LIN {X 0,Y 361.862,Z 339.034,A -85,B 0,C 180,E1 -13100.973,E2 -13100.973} C_VEL
LIN {X 0,Y 361.867,Z 339.03,A -85,B 0,C 180,E1 -13104.655,E2 -13104.655} C_VEL
LIN {X 0,Y 361.829,Z 339.027,A -85,B 0,C 180,E1 -13108.37,E2 -13108.37} C_VEL
LIN {X 0,Y 361.857,Z 339.016,A -85,B 0,C 180,E1 -13110.952,E2 -13110.952} C_VEL
LIN {X 0,Y 361.874,Z 339.028,A -85,B 0,C 180,E1 -13114.706,E2 -13114.706} C_VEL
LIN {X 0,Y 361.851,Z 339.032,A -85,B 0,C 180,E1 -13118.345,E2 -13118.345} C_VEL
LIN {X 0,Y 361.911,Z 339.028,A -85,B 0,C 180,E1 -13122.085,E2 -13122.085} C_VEL
LIN {X 0,Y 361.951,Z 339.022,A -85,B 0,C 180,E1 -13125.38,E2 -13125.38} C_VEL
LIN {X 0,Y 361.95,Z 339.014,A -85,B 0,C 180,E1 -13128.804,E2 -13128.804} C_VEL
LIN {X 0,Y 362.066,Z 339.002,A -85,B 0,C 180,E1 -13132.191,E2 -13132.191} C_VEL
LIN {X 0,Y 362.08,Z 339.004,A -85,B 0,C 180,E1 -13134.431,E2 -13134.431} C_VEL
LIN {X 0,Y 362.253,Z 338.978,A -85,B 0,C 180,E1 -13137.777,E2 -13137.777} C_VEL
LIN {X 0,Y 362.26,Z 338.976,A -85,B 0,C 180,E1 -13142.224,E2 -13142.224} C_VEL
LIN {X 0,Y 362.131,Z 338.998,A -85,B 0,C 180,E1 -13146.687,E2 -13146.687} C_VEL
LIN {X 0,Y 361.989,Z 339.017,A -85,B 0,C 180,E1 -13150.064,E2 -13150.064} C_VEL
LIN {X 0,Y 361.989,Z 339.017,A -85,B 0,C 180,E1 -13153.899,E2 -13153.899} C_VEL
LIN {X 0,Y 361.919,Z 339.022,A -85,B 0,C 180,E1 -13156.935,E2 -13156.935} C_VEL
LIN {X 0,Y 361.875,Z 339.028,A -85,B 0,C 180,E1 -13160.462,E2 -13160.462} C_VEL
LIN {X 0,Y 361.886,Z 339.028,A -85,B 0,C 180,E1 -13164.114,E2 -13164.114} C_VEL
LIN {X 0,Y 361.935,Z 339.028,A -85,B 0,C 180,E1 -13166.722,E2 -13166.722} C_VEL
LIN {X 0,Y 361.867,Z 339.035,A -85,B 0,C 180,E1 -13170.329,E2 -13170.329} C_VEL
LIN {X 0,Y 361.849,Z 339.033,A -85,B 0,C 180,E1 -13174.282,E2 -13174.282} C_VEL
LIN {X 0,Y 361.858,Z 339.029,A -85,B 0,C 180,E1 -13177.224,E2 -13177.224} C_VEL
LIN {X 0,Y 361.831,Z 339.038,A -85,B 0,C 180,E1 -13180.756,E2 -13180.756} C_VEL
LIN {X 0,Y 361.814,Z 339.041,A -85,B 0,C 180,E1 -13184.37,E2 -13184.37} C_VEL
LIN {X 0,Y 361.834,Z 339.039,A -85,B 0,C 180,E1 -13187.569,E2 -13187.569} C_VEL
LIN {X 0,Y 361.87,Z 339.036,A -85,B 0,C 180,E1 -13190.974,E2 -13190.974} C_VEL
LIN {X 0,Y 361.896,Z 339.076,A -85,B 0,C 180,E1 -13193.507,E2 -13193.507} C_VEL
LIN {X 0,Y 364.21,Z 348.551,A -85,B 0,C 180,E1 -13196.226,E2 -13196.226} C_VEL
LIN {X 0,Y 374.313,Z 370.595,A -85,B 0,C 180,E1 -13197.6,E2 -13197.6} C_VEL
LIN {X 0,Y 376.246,Z 375.985,A -85,B 0,C 180,E1 -13197.878,E2 -13197.878} C_VEL
LIN {X 0,Y 377.03,Z 379.634,A -85,B 0,C 180,E1 -13198.02,E2 -13198.02} C_VEL
LIN {X 0,Y 374.531,Z 484.966,A -85,B 0,C 180,E1 -13200.078,E2 -13200.078} C_VEL
LIN {X 0,Y 373.805,Z 499.549,A -85,B 0,C 180,E1 -13200.585,E2 -13200.585} C_VEL
LIN {X 0,Y 372.836,Z 513.064,A -85,B 0,C 180,E1 -13201.271,E2 -13201.271} C_VEL
LIN {X 0,Y 371.435,Z 527.178,A -85,B 0,C 180,E1 -13202.23,E2 -13202.23} C_VEL
LIN {X 0,Y 369.952,Z 539.936,A -85,B 0,C 180,E1 -13203.353,E2 -13203.353} C_VEL
LIN {X 0,Y 368.362,Z 551.192,A -85,B 0,C 180,E1 -13204.579,E2 -13204.579} C_VEL
LIN {X 0,Y 366.879,Z 561.686,A -85,B 0,C 180,E1 -13205.98,E2 -13205.98} C_VEL
LIN {X 0,Y 365.475,Z 572.081,A -85,B 0,C 180,E1 -13207.68,E2 -13207.68} C_VEL
LIN {X 0,Y 364.078,Z 580.622,A -85,B 0,C 180,E1 -13209.373,E2 -13209.373} C_VEL
LIN {X 0,Y 362.866,Z 588.744,A -85,B 0,C 180,E1 -13211.364,E2 -13211.364} C_VEL
LIN {X 0,Y 362.032,Z 594.441,A -85,B 0,C 180,E1 -13213.071,E2 -13213.071} C_VEL
LIN {X 0,Y 361.23,Z 600.377,A -85,B 0,C 180,E1 -13215.35,E2 -13215.35} C_VEL
LIN {X 0,Y 360.7,Z 604.706,A -85,B 0,C 180,E1 -13217.624,E2 -13217.624} C_VEL
LIN {X 0,Y 360.32,Z 607.567,A -85,B 0,C 180,E1 -13219.89,E2 -13219.89} C_VEL
LIN {X 0,Y 360.302,Z 609.048,A -85,B 0,C 180,E1 -13222.152,E2 -13222.152} C_VEL
LIN {X 0,Y 360.342,Z 609.198,A -85,B 0,C 180,E1 -13224.404,E2 -13224.404} C_VEL
LIN {X 0,Y 360.318,Z 608.032,A -85,B 0,C 180,E1 -13226.646,E2 -13226.646} C_VEL
LIN {X 0,Y 360.47,Z 605.531,A -85,B 0,C 180,E1 -13228.883,E2 -13228.883} C_VEL
LIN {X 0,Y 360.675,Z 601.614,A -85,B 0,C 180,E1 -13231.116,E2 -13231.116} C_VEL
LIN {X 0,Y 361.122,Z 596.159,A -85,B 0,C 180,E1 -13233.347,E2 -13233.347} C_VEL
LIN {X 0,Y 361.799,Z 589.999,A -85,B 0,C 180,E1 -13235.294,E2 -13235.294} C_VEL
LIN {X 0,Y 362.798,Z 582.325,A -85,B 0,C 180,E1 -13237.233,E2 -13237.233} C_VEL
LIN {X 0,Y 363.83,Z 574.327,A -85,B 0,C 180,E1 -13238.889,E2 -13238.889} C_VEL
LIN {X 0,Y 364.883,Z 564.682,A -85,B 0,C 180,E1 -13240.548,E2 -13240.548} C_VEL
LIN {X 0,Y 366.129,Z 554.042,A -85,B 0,C 180,E1 -13242.049,E2 -13242.049} C_VEL
LIN {X 0,Y 367.506,Z 542.214,A -85,B 0,C 180,E1 -13243.407,E2 -13243.407} C_VEL
LIN {X 0,Y 368.64,Z 530.605,A -85,B 0,C 180,E1 -13244.49,E2 -13244.49} C_VEL
LIN {X 0,Y 369.853,Z 516.946,A -85,B 0,C 180,E1 -13245.498,E2 -13245.498} C_VEL
LIN {X 0,Y 370.304,Z 510.93,A -85,B 0,C 180,E1 -13245.859,E2 -13245.859} C_VEL
LIN {X 0,Y 370.012,Z 505.422,A -85,B 0,C 180,E1 -13246.193,E2 -13246.193} C_VEL
LIN {X 0,Y 367.793,Z 496.434,A -85,B 0,C 180,E1 -13246.755,E2 -13246.755} C_VEL
LIN {X 0,Y 365.53,Z 487.277,A -85,B 0,C 180,E1 -13247.225,E2 -13247.225} C_VEL
LIN {X 0,Y 365.142,Z 481.513,A -85,B 0,C 180,E1 -13247.408,E2 -13247.408} C_VEL
LIN {X 0,Y 367.072,Z 379.114,A -85,B 0,C 180,E1 -13249.428,E2 -13249.428} C_VEL
LIN {X 0,Y 365.066,Z 369.722,A -85,B 0,C 180,E1 -13249.762,E2 -13249.762} C_VEL
LIN {X 0,Y 357.701,Z 350.958,A -85,B 0,C 180,E1 -13250.685,E2 -13250.685} C_VEL
LIN {X 0,Y 356.686,Z 348.279,A -85,B 0,C 180,E1 -13250.833,E2 -13250.833} C_VEL
LIN {X 0,Y 354.849,Z 339.909,A -85,B 0,C 180,E1 -13253.142,E2 -13253.142} C_VEL
LIN {X 0,Y 354.889,Z 339.904,A -85,B 0,C 180,E1 -13256.98,E2 -13256.98} C_VEL
LIN {X 0,Y 354.819,Z 339.911,A -85,B 0,C 180,E1 -13259.681,E2 -13259.681} C_VEL
LIN {X 0,Y 354.806,Z 339.916,A -85,B 0,C 180,E1 -13263.701,E2 -13263.701} C_VEL
LIN {X 0,Y 354.801,Z 339.91,A -85,B 0,C 180,E1 -13266.458,E2 -13266.458} C_VEL
LIN {X 0,Y 354.823,Z 339.901,A -85,B 0,C 180,E1 -13269.422,E2 -13269.422} C_VEL
LIN {X 0,Y 354.786,Z 339.914,A -85,B 0,C 180,E1 -13272.866,E2 -13272.866} C_VEL
LIN {X 0,Y 354.764,Z 339.918,A -85,B 0,C 180,E1 -13276.102,E2 -13276.102} C_VEL
LIN {X 0,Y 354.783,Z 339.913,A -85,B 0,C 180,E1 -13279.178,E2 -13279.178} C_VEL
LIN {X 0,Y 354.802,Z 339.906,A -85,B 0,C 180,E1 -13282.402,E2 -13282.402} C_VEL
LIN {X 0,Y 354.807,Z 339.915,A -85,B 0,C 180,E1 -13284.94,E2 -13284.94} C_VEL
LIN {X 0,Y 354.787,Z 339.913,A -85,B 0,C 180,E1 -13288.404,E2 -13288.404} C_VEL
LIN {X 0,Y 354.831,Z 339.898,A -85,B 0,C 180,E1 -13291.617,E2 -13291.617} C_VEL
LIN {X 0,Y 354.867,Z 339.899,A -85,B 0,C 180,E1 -13294.17,E2 -13294.17} C_VEL
LIN {X 0,Y 354.8,Z 339.907,A -85,B 0,C 180,E1 -13297.891,E2 -13297.891} C_VEL
LIN {X 0,Y 354.881,Z 339.899,A -85,B 0,C 180,E1 -13301.907,E2 -13301.907} C_VEL
LIN {X 0,Y 354.934,Z 339.888,A -85,B 0,C 180,E1 -13305.981,E2 -13305.981} C_VEL
LIN {X 0,Y 354.945,Z 339.89,A -85,B 0,C 180,E1 -13309.734,E2 -13309.734} C_VEL
LIN {X 0,Y 355.095,Z 339.87,A -85,B 0,C 180,E1 -13313.18,E2 -13313.18} C_VEL
LIN {X 0,Y 355.219,Z 339.855,A -85,B 0,C 180,E1 -13317.732,E2 -13317.732} C_VEL
LIN {X 0,Y 355.159,Z 339.864,A -85,B 0,C 180,E1 -13321.133,E2 -13321.133} C_VEL
LIN {X 0,Y 355.206,Z 339.856,A -85,B 0,C 180,E1 -13322.267,E2 -13322.267} C_VEL
LIN {X 0,Y 355.073,Z 339.879,A -85,B 0,C 180,E1 -13326.82,E2 -13326.82} C_VEL
LIN {X 0,Y 354.943,Z 339.887,A -85,B 0,C 180,E1 -13330.265,E2 -13330.265} C_VEL
LIN {X 0,Y 354.933,Z 339.897,A -85,B 0,C 180,E1 -13334.018,E2 -13334.018} C_VEL
LIN {X 0,Y 354.88,Z 339.904,A -85,B 0,C 180,E1 -13338.092,E2 -13338.092} C_VEL
LIN {X 0,Y 354.805,Z 339.906,A -85,B 0,C 180,E1 -13342.108,E2 -13342.108} C_VEL
LIN {X 0,Y 354.812,Z 339.906,A -85,B 0,C 180,E1 -13345.834,E2 -13345.834} C_VEL
LIN {X 0,Y 354.788,Z 339.914,A -85,B 0,C 180,E1 -13349.684,E2 -13349.684} C_VEL
LIN {X 0,Y 354.778,Z 339.917,A -85,B 0,C 180,E1 -13352.334,E2 -13352.334} C_VEL
LIN {X 0,Y 354.814,Z 339.914,A -85,B 0,C 180,E1 -13355.7,E2 -13355.7} C_VEL
LIN {X 0,Y 354.817,Z 339.913,A -85,B 0,C 180,E1 -13359.424,E2 -13359.424} C_VEL
LIN {X 0,Y 354.782,Z 339.912,A -85,B 0,C 180,E1 -13362.868,E2 -13362.868} C_VEL
LIN {X 0,Y 354.761,Z 339.919,A -85,B 0,C 180,E1 -13366.104,E2 -13366.104} C_VEL
LIN {X 0,Y 354.782,Z 339.918,A -85,B 0,C 180,E1 -13369.18,E2 -13369.18} C_VEL
LIN {X 0,Y 354.802,Z 339.918,A -85,B 0,C 180,E1 -13372.403,E2 -13372.403} C_VEL
LIN {X 0,Y 354.808,Z 339.919,A -85,B 0,C 180,E1 -13374.942,E2 -13374.942} C_VEL
LIN {X 0,Y 354.835,Z 340.014,A -85,B 0,C 180,E1 -13377.168,E2 -13377.168} C_VEL
LIN {X 0,Y 358.077,Z 353.914,A -85,B 0,C 180,E1 -13380.616,E2 -13380.616} C_VEL
LIN {X 0,Y 360.084,Z 364.069,A -85,B 0,C 180,E1 -13383.014,E2 -13383.014} C_VEL
LIN {X 0,Y 360.134,Z 366.037,A -85,B 0,C 180,E1 -13383.448,E2 -13383.448} C_VEL
LIN {X 0,Y 365.056,Z 394.772,A -85,B 0,C 180,E1 -13384.402,E2 -13384.402} C_VEL
LIN {X 0,Y 366.748,Z 405.34,A -85,B 0,C 180,E1 -13384.736,E2 -13384.736} C_VEL
LIN {X 0,Y 364.738,Z 503.037,A -85,B 0,C 180,E1 -13386.659,E2 -13386.659} C_VEL
LIN {X 0,Y 364,Z 517.441,A -85,B 0,C 180,E1 -13387.135,E2 -13387.135} C_VEL
LIN {X 0,Y 363.018,Z 531.264,A -85,B 0,C 180,E1 -13387.821,E2 -13387.821} C_VEL
LIN {X 0,Y 361.901,Z 543.849,A -85,B 0,C 180,E1 -13388.655,E2 -13388.655} C_VEL
LIN {X 0,Y 360.585,Z 556.821,A -85,B 0,C 180,E1 -13389.76,E2 -13389.76} C_VEL
LIN {X 0,Y 359.18,Z 568.653,A -85,B 0,C 180,E1 -13391.017,E2 -13391.017} C_VEL
LIN {X 0,Y 357.972,Z 578.49,A -85,B 0,C 180,E1 -13392.284,E2 -13392.284} C_VEL
LIN {X 0,Y 356.588,Z 589.361,A -85,B 0,C 180,E1 -13393.983,E2 -13393.983} C_VEL
LIN {X 0,Y 355.57,Z 598.603,A -85,B 0,C 180,E1 -13395.753,E2 -13395.753} C_VEL
LIN {X 0,Y 354.694,Z 606.928,A -85,B 0,C 180,E1 -13397.702,E2 -13397.702} C_VEL
LIN {X 0,Y 353.92,Z 613.835,A -85,B 0,C 180,E1 -13399.705,E2 -13399.705} C_VEL
LIN {X 0,Y 353.58,Z 618.593,A -85,B 0,C 180,E1 -13401.427,E2 -13401.427} C_VEL
LIN {X 0,Y 353.4,Z 622.44,A -85,B 0,C 180,E1 -13403.147,E2 -13403.147} C_VEL
LIN {X 0,Y 353.269,Z 626.191,A -85,B 0,C 180,E1 -13405.436,E2 -13405.436} C_VEL
LIN {X 0,Y 353.181,Z 628.521,A -85,B 0,C 180,E1 -13407.719,E2 -13407.719} C_VEL
LIN {X 0,Y 353.261,Z 629.496,A -85,B 0,C 180,E1 -13410,E2 -13410} C_VEL
LIN {X 0,Y 353.168,Z 629.129,A -85,B 0,C 180,E1 -13412.281,E2 -13412.281} C_VEL
LIN {X 0,Y 353.246,Z 627.432,A -85,B 0,C 180,E1 -13414.564,E2 -13414.564} C_VEL
LIN {X 0,Y 353.411,Z 624.368,A -85,B 0,C 180,E1 -13416.853,E2 -13416.853} C_VEL
LIN {X 0,Y 353.772,Z 619.856,A -85,B 0,C 180,E1 -13419.144,E2 -13419.144} C_VEL
LIN {X 0,Y 354.219,Z 615.396,A -85,B 0,C 180,E1 -13420.864,E2 -13420.864} C_VEL
LIN {X 0,Y 355.178,Z 608.979,A -85,B 0,C 180,E1 -13422.862,E2 -13422.862} C_VEL
LIN {X 0,Y 356.2,Z 601.025,A -85,B 0,C 180,E1 -13424.862,E2 -13424.862} C_VEL
LIN {X 0,Y 357.49,Z 592.726,A -85,B 0,C 180,E1 -13426.562,E2 -13426.562} C_VEL
LIN {X 0,Y 359.067,Z 582.754,A -85,B 0,C 180,E1 -13428.25,E2 -13428.25} C_VEL
LIN {X 0,Y 360.864,Z 571.675,A -85,B 0,C 180,E1 -13429.778,E2 -13429.778} C_VEL
LIN {X 0,Y 362.613,Z 559.29,A -85,B 0,C 180,E1 -13431.16,E2 -13431.16} C_VEL
LIN {X 0,Y 364.133,Z 547.349,A -85,B 0,C 180,E1 -13432.231,E2 -13432.231} C_VEL
LIN {X 0,Y 365.442,Z 534.552,A -85,B 0,C 180,E1 -13433.143,E2 -13433.143} C_VEL
LIN {X 0,Y 366.783,Z 520.612,A -85,B 0,C 180,E1 -13433.877,E2 -13433.877} C_VEL
LIN {X 0,Y 367.758,Z 505.981,A -85,B 0,C 180,E1 -13434.409,E2 -13434.409} C_VEL
LIN {X 0,Y 368.551,Z 481.48,A -85,B 0,C 180,E1 -13434.928,E2 -13434.928} C_VEL
LIN {X 0,Y 370.194,Z 405.301,A -85,B 0,C 180,E1 -13436.436,E2 -13436.436} C_VEL
LIN {X 0,Y 365.616,Z 381.424,A -85,B 0,C 180,E1 -13437.353,E2 -13437.353} C_VEL
LIN {X 0,Y 362.959,Z 370.452,A -85,B 0,C 180,E1 -13437.836,E2 -13437.836} C_VEL
LIN {X 0,Y 361.045,Z 365.765,A -85,B 0,C 180,E1 -13438.117,E2 -13438.117} C_VEL
LIN {X 0,Y 358.588,Z 354.578,A -85,B 0,C 180,E1 -13440.961,E2 -13440.961} C_VEL
LIN {X 0,Y 355.383,Z 342.059,A -85,B 0,C 180,E1 -13444.354,E2 -13444.354} C_VEL
LIN {X 0,Y 354.869,Z 339.906,A -85,B 0,C 180,E1 -13444.971,E2 -13444.971} C_VEL
LIN {X 0,Y 354.801,Z 339.903,A -85,B 0,C 180,E1 -13447.882,E2 -13447.882} C_VEL
LIN {X 0,Y 354.782,Z 339.904,A -85,B 0,C 180,E1 -13451.171,E2 -13451.171} C_VEL
LIN {X 0,Y 354.758,Z 339.914,A -85,B 0,C 180,E1 -13454.506,E2 -13454.506} C_VEL
LIN {X 0,Y 354.788,Z 339.91,A -85,B 0,C 180,E1 -13457.662,E2 -13457.662} C_VEL
LIN {X 0,Y 354.809,Z 339.914,A -85,B 0,C 180,E1 -13460.665,E2 -13460.665} C_VEL
LIN {X 0,Y 354.814,Z 339.911,A -85,B 0,C 180,E1 -13464.3,E2 -13464.3} C_VEL
LIN {X 0,Y 354.779,Z 339.915,A -85,B 0,C 180,E1 -13467.666,E2 -13467.666} C_VEL
LIN {X 0,Y 354.793,Z 339.9,A -85,B 0,C 180,E1 -13471.614,E2 -13471.614} C_VEL
LIN {X 0,Y 354.825,Z 339.905,A -85,B 0,C 180,E1 -13475.657,E2 -13475.657} C_VEL
LIN {X 0,Y 354.816,Z 339.907,A -85,B 0,C 180,E1 -13479.113,E2 -13479.113} C_VEL
LIN {X 0,Y 354.87,Z 339.902,A -85,B 0,C 180,E1 -13482.719,E2 -13482.719} C_VEL
LIN {X 0,Y 354.941,Z 339.896,A -85,B 0,C 180,E1 -13486.255,E2 -13486.255} C_VEL
LIN {X 0,Y 354.939,Z 339.896,A -85,B 0,C 180,E1 -13489.735,E2 -13489.735} C_VEL
LIN {X 0,Y 355.076,Z 339.871,A -85,B 0,C 180,E1 -13493.18,E2 -13493.18} C_VEL
LIN {X 0,Y 355.216,Z 339.854,A -85,B 0,C 180,E1 -13497.733,E2 -13497.733} C_VEL
LIN {X 0,Y 355.223,Z 339.853,A -85,B 0,C 180,E1 -13502.268,E2 -13502.268} C_VEL
LIN {X 0,Y 355.095,Z 339.873,A -85,B 0,C 180,E1 -13506.82,E2 -13506.82} C_VEL
LIN {X 0,Y 354.945,Z 339.895,A -85,B 0,C 180,E1 -13510.265,E2 -13510.265} C_VEL
LIN {X 0,Y 354.934,Z 339.896,A -85,B 0,C 180,E1 -13514.019,E2 -13514.019} C_VEL
LIN {X 0,Y 354.882,Z 339.902,A -85,B 0,C 180,E1 -13518.093,E2 -13518.093} C_VEL
LIN {X 0,Y 354.809,Z 339.911,A -85,B 0,C 180,E1 -13522.108,E2 -13522.108} C_VEL
LIN {X 0,Y 354.892,Z 339.901,A -85,B 0,C 180,E1 -13525.829,E2 -13525.829} C_VEL
LIN {X 0,Y 354.812,Z 339.912,A -85,B 0,C 180,E1 -13529.683,E2 -13529.683} C_VEL
LIN {X 0,Y 354.801,Z 339.911,A -85,B 0,C 180,E1 -13533.703,E2 -13533.703} C_VEL
LIN {X 0,Y 354.793,Z 339.915,A -85,B 0,C 180,E1 -13536.461,E2 -13536.461} C_VEL
LIN {X 0,Y 354.821,Z 339.908,A -85,B 0,C 180,E1 -13539.425,E2 -13539.425} C_VEL
LIN {X 0,Y 354.785,Z 339.915,A -85,B 0,C 180,E1 -13542.868,E2 -13542.868} C_VEL
LIN {X 0,Y 354.765,Z 339.922,A -85,B 0,C 180,E1 -13546.105,E2 -13546.105} C_VEL
LIN {X 0,Y 354.787,Z 339.917,A -85,B 0,C 180,E1 -13549.18,E2 -13549.18} C_VEL
LIN {X 0,Y 354.864,Z 340.034,A -85,B 0,C 180,E1 -13552.974,E2 -13552.974} C_VEL
LIN {X 0,Y 357.101,Z 348.911,A -85,B 0,C 180,E1 -13555.565,E2 -13555.565} C_VEL
LIN {X 0,Y 368.009,Z 372.395,A -85,B 0,C 180,E1 -13557.097,E2 -13557.097} C_VEL
LIN {X 0,Y 370.229,Z 378.271,A -85,B 0,C 180,E1 -13557.418,E2 -13557.418} C_VEL
LIN {X 0,Y 370.796,Z 381.796,A -85,B 0,C 180,E1 -13557.543,E2 -13557.543} C_VEL
LIN {X 0,Y 368.182,Z 485.531,A -85,B 0,C 180,E1 -13559.603,E2 -13559.603} C_VEL
LIN {X 0,Y 367.435,Z 499.771,A -85,B 0,C 180,E1 -13560.108,E2 -13560.108} C_VEL
LIN {X 0,Y 366.413,Z 513.206,A -85,B 0,C 180,E1 -13560.798,E2 -13560.798} C_VEL
LIN {X 0,Y 365.051,Z 526.435,A -85,B 0,C 180,E1 -13561.701,E2 -13561.701} C_VEL
LIN {X 0,Y 363.51,Z 539.377,A -85,B 0,C 180,E1 -13562.842,E2 -13562.842} C_VEL
LIN {X 0,Y 361.829,Z 550.767,A -85,B 0,C 180,E1 -13564.086,E2 -13564.086} C_VEL
LIN {X 0,Y 360.262,Z 561.366,A -85,B 0,C 180,E1 -13565.51,E2 -13565.51} C_VEL
LIN {X 0,Y 358.845,Z 571.348,A -85,B 0,C 180,E1 -13567.149,E2 -13567.149} C_VEL
LIN {X 0,Y 357.315,Z 580.481,A -85,B 0,C 180,E1 -13568.964,E2 -13568.964} C_VEL
LIN {X 0,Y 356.017,Z 588.676,A -85,B 0,C 180,E1 -13570.992,E2 -13570.992} C_VEL
LIN {X 0,Y 355.102,Z 594.414,A -85,B 0,C 180,E1 -13572.731,E2 -13572.731} C_VEL
LIN {X 0,Y 354.4,Z 599.061,A -85,B 0,C 180,E1 -13574.472,E2 -13574.472} C_VEL
LIN {X 0,Y 353.824,Z 603.737,A -85,B 0,C 180,E1 -13576.73,E2 -13576.73} C_VEL
LIN {X 0,Y 353.453,Z 606.418,A -85,B 0,C 180,E1 -13578.531,E2 -13578.531} C_VEL
LIN {X 0,Y 353.211,Z 608.625,A -85,B 0,C 180,E1 -13580.841,E2 -13580.841} C_VEL
LIN {X 0,Y 353.235,Z 609.479,A -85,B 0,C 180,E1 -13583.144,E2 -13583.144} C_VEL
LIN {X 0,Y 353.255,Z 609.013,A -85,B 0,C 180,E1 -13585.436,E2 -13585.436} C_VEL
LIN {X 0,Y 353.256,Z 607.229,A -85,B 0,C 180,E1 -13587.72,E2 -13587.72} C_VEL
LIN {X 0,Y 353.496,Z 604.088,A -85,B 0,C 180,E1 -13590,E2 -13590} C_VEL
LIN {X 0,Y 353.782,Z 599.478,A -85,B 0,C 180,E1 -13592.277,E2 -13592.277} C_VEL
LIN {X 0,Y 354.436,Z 593.245,A -85,B 0,C 180,E1 -13594.549,E2 -13594.549} C_VEL
LIN {X 0,Y 355.346,Z 586.307,A -85,B 0,C 180,E1 -13596.53,E2 -13596.53} C_VEL
LIN {X 0,Y 356.485,Z 577.725,A -85,B 0,C 180,E1 -13598.503,E2 -13598.503} C_VEL
LIN {X 0,Y 357.488,Z 568.775,A -85,B 0,C 180,E1 -13600.191,E2 -13600.191} C_VEL
LIN {X 0,Y 358.818,Z 558.319,A -85,B 0,C 180,E1 -13601.81,E2 -13601.81} C_VEL
LIN {X 0,Y 360.221,Z 546.912,A -85,B 0,C 180,E1 -13603.252,E2 -13603.252} C_VEL
LIN {X 0,Y 361.491,Z 534.771,A -85,B 0,C 180,E1 -13604.496,E2 -13604.496} C_VEL
LIN {X 0,Y 362.784,Z 521.16,A -85,B 0,C 180,E1 -13605.592,E2 -13605.592} C_VEL
LIN {X 0,Y 363.879,Z 507.894,A -85,B 0,C 180,E1 -13606.407,E2 -13606.407} C_VEL
LIN {X 0,Y 364.735,Z 493.425,A -85,B 0,C 180,E1 -13607.052,E2 -13607.052} C_VEL
LIN {X 0,Y 365.142,Z 481.513,A -85,B 0,C 180,E1 -13607.408,E2 -13607.408} C_VEL
LIN {X 0,Y 364.716,Z 475.716,A -85,B 0,C 180,E1 -13607.571,E2 -13607.571} C_VEL
LIN {X 0,Y 359.648,Z 457.052,A -85,B 0,C 180,E1 -13608.283,E2 -13608.283} C_VEL
LIN {X 0,Y 359.123,Z 451.241,A -85,B 0,C 180,E1 -13608.438,E2 -13608.438} C_VEL
LIN {X 0,Y 360.597,Z 380.281,A -85,B 0,C 180,E1 -13609.848,E2 -13609.848} C_VEL
LIN {X 0,Y 358.726,Z 371.861,A -85,B 0,C 180,E1 -13610.16,E2 -13610.16} C_VEL
LIN {X 0,Y 351.347,Z 353.141,A -85,B 0,C 180,E1 -13611.111,E2 -13611.111} C_VEL
LIN {X 0,Y 349.48,Z 348.49,A -85,B 0,C 180,E1 -13611.373,E2 -13611.373} C_VEL
LIN {X 0,Y 347.804,Z 340.788,A -85,B 0,C 180,E1 -13613.52,E2 -13613.52} C_VEL
LIN {X 0,Y 347.852,Z 340.781,A -85,B 0,C 180,E1 -13617.254,E2 -13617.254} C_VEL
LIN {X 0,Y 347.75,Z 340.793,A -85,B 0,C 180,E1 -13620.347,E2 -13620.347} C_VEL
LIN {X 0,Y 347.749,Z 340.792,A -85,B 0,C 180,E1 -13624.043,E2 -13624.043} C_VEL
LIN {X 0,Y 347.765,Z 340.79,A -85,B 0,C 180,E1 -13627.319,E2 -13627.319} C_VEL
LIN {X 0,Y 347.73,Z 340.777,A -85,B 0,C 180,E1 -13630.296,E2 -13630.296} C_VEL
LIN {X 0,Y 347.721,Z 340.799,A -85,B 0,C 180,E1 -13633.407,E2 -13633.407} C_VEL
LIN {X 0,Y 347.722,Z 340.795,A -85,B 0,C 180,E1 -13636.685,E2 -13636.685} C_VEL
LIN {X 0,Y 347.743,Z 340.792,A -85,B 0,C 180,E1 -13640.172,E2 -13640.172} C_VEL
LIN {X 0,Y 347.756,Z 340.784,A -85,B 0,C 180,E1 -13642.678,E2 -13642.678} C_VEL
LIN {X 0,Y 347.743,Z 340.787,A -85,B 0,C 180,E1 -13645.955,E2 -13645.955} C_VEL
LIN {X 0,Y 347.743,Z 340.792,A -85,B 0,C 180,E1 -13649.651,E2 -13649.651} C_VEL
LIN {X 0,Y 347.804,Z 340.778,A -85,B 0,C 180,E1 -13653.605,E2 -13653.605} C_VEL
LIN {X 0,Y 347.774,Z 340.788,A -85,B 0,C 180,E1 -13656.16,E2 -13656.16} C_VEL
LIN {X 0,Y 347.777,Z 340.771,A -85,B 0,C 180,E1 -13659.907,E2 -13659.907} C_VEL
LIN {X 0,Y 347.823,Z 340.781,A -85,B 0,C 180,E1 -13663.567,E2 -13663.567} C_VEL
LIN {X 0,Y 347.879,Z 340.757,A -85,B 0,C 180,E1 -13667.16,E2 -13667.16} C_VEL
LIN {X 0,Y 347.925,Z 340.771,A -85,B 0,C 180,E1 -13670.7,E2 -13670.7} C_VEL
LIN {X 0,Y 348.062,Z 340.747,A -85,B 0,C 180,E1 -13673.041,E2 -13673.041} C_VEL
LIN {X 0,Y 348.181,Z 340.732,A -85,B 0,C 180,E1 -13677.686,E2 -13677.686} C_VEL
LIN {X 0,Y 348.128,Z 340.74,A -85,B 0,C 180,E1 -13681.156,E2 -13681.156} C_VEL
LIN {X 0,Y 348.143,Z 340.734,A -85,B 0,C 180,E1 -13682.314,E2 -13682.314} C_VEL
LIN {X 0,Y 348.04,Z 340.754,A -85,B 0,C 180,E1 -13686.959,E2 -13686.959} C_VEL
LIN {X 0,Y 347.883,Z 340.768,A -85,B 0,C 180,E1 -13690.475,E2 -13690.475} C_VEL
LIN {X 0,Y 347.889,Z 340.772,A -85,B 0,C 180,E1 -13694.15,E2 -13694.15} C_VEL
LIN {X 0,Y 347.819,Z 340.786,A -85,B 0,C 180,E1 -13698.259,E2 -13698.259} C_VEL
LIN {X 0,Y 347.758,Z 340.779,A -85,B 0,C 180,E1 -13701.626,E2 -13701.626} C_VEL
LIN {X 0,Y 347.764,Z 340.784,A -85,B 0,C 180,E1 -13705.112,E2 -13705.112} C_VEL
LIN {X 0,Y 347.73,Z 340.792,A -85,B 0,C 180,E1 -13707.701,E2 -13707.701} C_VEL
LIN {X 0,Y 347.73,Z 340.789,A -85,B 0,C 180,E1 -13710.349,E2 -13710.349} C_VEL
LIN {X 0,Y 347.741,Z 340.791,A -85,B 0,C 180,E1 -13714.044,E2 -13714.044} C_VEL
LIN {X 0,Y 347.754,Z 340.79,A -85,B 0,C 180,E1 -13717.321,E2 -13717.321} C_VEL
LIN {X 0,Y 347.725,Z 340.788,A -85,B 0,C 180,E1 -13720.298,E2 -13720.298} C_VEL
LIN {X 0,Y 347.717,Z 340.795,A -85,B 0,C 180,E1 -13723.409,E2 -13723.409} C_VEL
LIN {X 0,Y 347.72,Z 340.794,A -85,B 0,C 180,E1 -13726.687,E2 -13726.687} C_VEL
LIN {X 0,Y 347.742,Z 340.797,A -85,B 0,C 180,E1 -13730.174,E2 -13730.174} C_VEL
LIN {X 0,Y 347.757,Z 340.796,A -85,B 0,C 180,E1 -13732.68,E2 -13732.68} C_VEL
LIN {X 0,Y 347.745,Z 340.797,A -85,B 0,C 180,E1 -13735.957,E2 -13735.957} C_VEL
LIN {X 0,Y 347.778,Z 340.857,A -85,B 0,C 180,E1 -13736.731,E2 -13736.731} C_VEL
LIN {X 0,Y 351.087,Z 354.883,A -85,B 0,C 180,E1 -13740.302,E2 -13740.302} C_VEL
LIN {X 0,Y 353.248,Z 365.981,A -85,B 0,C 180,E1 -13742.952,E2 -13742.952} C_VEL
LIN {X 0,Y 357.451,Z 388.861,A -85,B 0,C 180,E1 -13743.753,E2 -13743.753} C_VEL
LIN {X 0,Y 360.196,Z 405.899,A -85,B 0,C 180,E1 -13744.308,E2 -13744.308} C_VEL
LIN {X 0,Y 358.138,Z 502.445,A -85,B 0,C 180,E1 -13746.241,E2 -13746.241} C_VEL
LIN {X 0,Y 357.389,Z 517.036,A -85,B 0,C 180,E1 -13746.726,E2 -13746.726} C_VEL
LIN {X 0,Y 356.308,Z 531.485,A -85,B 0,C 180,E1 -13747.457,E2 -13747.457} C_VEL
LIN {X 0,Y 355.157,Z 544.008,A -85,B 0,C 180,E1 -13748.308,E2 -13748.308} C_VEL
LIN {X 0,Y 353.91,Z 556.17,A -85,B 0,C 180,E1 -13749.361,E2 -13749.361} C_VEL
LIN {X 0,Y 352.405,Z 568.079,A -85,B 0,C 180,E1 -13750.638,E2 -13750.638} C_VEL
LIN {X 0,Y 351.136,Z 577.98,A -85,B 0,C 180,E1 -13751.927,E2 -13751.927} C_VEL
LIN {X 0,Y 349.703,Z 588.904,A -85,B 0,C 180,E1 -13753.659,E2 -13753.659} C_VEL
LIN {X 0,Y 348.686,Z 597.64,A -85,B 0,C 180,E1 -13755.346,E2 -13755.346} C_VEL
LIN {X 0,Y 347.791,Z 605.421,A -85,B 0,C 180,E1 -13757.157,E2 -13757.157} C_VEL
LIN {X 0,Y 347.079,Z 611.662,A -85,B 0,C 180,E1 -13758.909,E2 -13758.909} C_VEL
LIN {X 0,Y 346.509,Z 618.281,A -85,B 0,C 180,E1 -13761.251,E2 -13761.251} C_VEL
LIN {X 0,Y 346.324,Z 622.156,A -85,B 0,C 180,E1 -13763.007,E2 -13763.007} C_VEL
LIN {X 0,Y 346.168,Z 625.934,A -85,B 0,C 180,E1 -13765.342,E2 -13765.342} C_VEL
LIN {X 0,Y 346.091,Z 628.289,A -85,B 0,C 180,E1 -13767.672,E2 -13767.672} C_VEL
LIN {X 0,Y 346.163,Z 629.288,A -85,B 0,C 180,E1 -13770,E2 -13770} C_VEL
LIN {X 0,Y 346.079,Z 628.946,A -85,B 0,C 180,E1 -13772.328,E2 -13772.328} C_VEL
LIN {X 0,Y 346.146,Z 627.273,A -85,B 0,C 180,E1 -13774.658,E2 -13774.658} C_VEL
LIN {X 0,Y 346.336,Z 624.234,A -85,B 0,C 180,E1 -13776.993,E2 -13776.993} C_VEL
LIN {X 0,Y 346.718,Z 619.748,A -85,B 0,C 180,E1 -13779.332,E2 -13779.332} C_VEL
LIN {X 0,Y 347.194,Z 615.317,A -85,B 0,C 180,E1 -13781.087,E2 -13781.087} C_VEL
LIN {X 0,Y 348.231,Z 608.933,A -85,B 0,C 180,E1 -13783.123,E2 -13783.123} C_VEL
LIN {X 0,Y 349.299,Z 601.014,A -85,B 0,C 180,E1 -13785.162,E2 -13785.162} C_VEL
LIN {X 0,Y 350.678,Z 592.756,A -85,B 0,C 180,E1 -13786.893,E2 -13786.893} C_VEL
LIN {X 0,Y 352.314,Z 582.83,A -85,B 0,C 180,E1 -13788.612,E2 -13788.612} C_VEL
LIN {X 0,Y 354.19,Z 571.813,A -85,B 0,C 180,E1 -13790.167,E2 -13790.167} C_VEL
LIN {X 0,Y 356.01,Z 559.537,A -85,B 0,C 180,E1 -13791.572,E2 -13791.572} C_VEL
LIN {X 0,Y 357.618,Z 547.402,A -85,B 0,C 180,E1 -13792.685,E2 -13792.685} C_VEL
LIN {X 0,Y 359.06,Z 533.942,A -85,B 0,C 180,E1 -13793.656,E2 -13793.656} C_VEL
LIN {X 0,Y 360.452,Z 519.863,A -85,B 0,C 180,E1 -13794.399,E2 -13794.399} C_VEL
LIN {X 0,Y 361.421,Z 506.091,A -85,B 0,C 180,E1 -13794.904,E2 -13794.904} C_VEL
LIN {X 0,Y 362.198,Z 483.438,A -85,B 0,C 180,E1 -13795.398,E2 -13795.398} C_VEL
LIN {X 0,Y 363.952,Z 406.151,A -85,B 0,C 180,E1 -13796.952,E2 -13796.952} C_VEL
LIN {X 0,Y 358.844,Z 379.915,A -85,B 0,C 180,E1 -13798,E2 -13798} C_VEL
LIN {X 0,Y 357.023,Z 372.931,A -85,B 0,C 180,E1 -13798.33,E2 -13798.33} C_VEL
LIN {X 0,Y 353.847,Z 365.477,A -85,B 0,C 180,E1 -13798.816,E2 -13798.816} C_VEL
LIN {X 0,Y 351.326,Z 354.695,A -85,B 0,C 180,E1 -13801.658,E2 -13801.658} C_VEL
LIN {X 0,Y 348.533,Z 343.682,A -85,B 0,C 180,E1 -13804.725,E2 -13804.725} C_VEL
LIN {X 0,Y 347.784,Z 340.787,A -85,B 0,C 180,E1 -13805.607,E2 -13805.607} C_VEL
LIN {X 0,Y 347.748,Z 340.789,A -85,B 0,C 180,E1 -13808.792,E2 -13808.792} C_VEL
LIN {X 0,Y 347.745,Z 340.786,A -85,B 0,C 180,E1 -13811.83,E2 -13811.83} C_VEL
LIN {X 0,Y 347.7,Z 340.79,A -85,B 0,C 180,E1 -13815.026,E2 -13815.026} C_VEL
LIN {X 0,Y 347.744,Z 340.794,A -85,B 0,C 180,E1 -13818.397,E2 -13818.397} C_VEL
LIN {X 0,Y 347.766,Z 340.789,A -85,B 0,C 180,E1 -13822.011,E2 -13822.011} C_VEL
LIN {X 0,Y 347.737,Z 340.789,A -85,B 0,C 180,E1 -13825.536,E2 -13825.536} C_VEL
LIN {X 0,Y 347.736,Z 340.783,A -85,B 0,C 180,E1 -13828.3,E2 -13828.3} C_VEL
LIN {X 0,Y 347.737,Z 340.773,A -85,B 0,C 180,E1 -13830.984,E2 -13830.984} C_VEL
LIN {X 0,Y 347.742,Z 340.794,A -85,B 0,C 180,E1 -13833.601,E2 -13833.601} C_VEL
LIN {X 0,Y 347.76,Z 340.788,A -85,B 0,C 180,E1 -13836.16,E2 -13836.16} C_VEL
LIN {X 0,Y 347.788,Z 340.782,A -85,B 0,C 180,E1 -13839.908,E2 -13839.908} C_VEL
LIN {X 0,Y 347.821,Z 340.777,A -85,B 0,C 180,E1 -13843.568,E2 -13843.568} C_VEL
LIN {X 0,Y 347.875,Z 340.776,A -85,B 0,C 180,E1 -13847.16,E2 -13847.16} C_VEL
LIN {X 0,Y 347.923,Z 340.77,A -85,B 0,C 180,E1 -13850.701,E2 -13850.701} C_VEL
LIN {X 0,Y 348.028,Z 340.755,A -85,B 0,C 180,E1 -13854.205,E2 -13854.205} C_VEL
LIN {X 0,Y 348.177,Z 340.73,A -85,B 0,C 180,E1 -13857.687,E2 -13857.687} C_VEL
LIN {X 0,Y 348.106,Z 340.748,A -85,B 0,C 180,E1 -13861.157,E2 -13861.157} C_VEL
LIN {X 0,Y 348.184,Z 340.729,A -85,B 0,C 180,E1 -13862.314,E2 -13862.314} C_VEL
LIN {X 0,Y 348.062,Z 340.747,A -85,B 0,C 180,E1 -13866.959,E2 -13866.959} C_VEL
LIN {X 0,Y 347.886,Z 340.775,A -85,B 0,C 180,E1 -13870.476,E2 -13870.476} C_VEL
LIN {X 0,Y 347.891,Z 340.774,A -85,B 0,C 180,E1 -13874.151,E2 -13874.151} C_VEL
LIN {X 0,Y 347.821,Z 340.782,A -85,B 0,C 180,E1 -13878.26,E2 -13878.26} C_VEL
LIN {X 0,Y 347.761,Z 340.789,A -85,B 0,C 180,E1 -13881.627,E2 -13881.627} C_VEL
LIN {X 0,Y 347.805,Z 340.783,A -85,B 0,C 180,E1 -13885.11,E2 -13885.11} C_VEL
LIN {X 0,Y 347.802,Z 340.78,A -85,B 0,C 180,E1 -13887.695,E2 -13887.695} C_VEL
LIN {X 0,Y 347.743,Z 340.795,A -85,B 0,C 180,E1 -13890.349,E2 -13890.349} C_VEL
LIN {X 0,Y 347.743,Z 340.791,A -85,B 0,C 180,E1 -13894.045,E2 -13894.045} C_VEL
LIN {X 0,Y 347.757,Z 340.785,A -85,B 0,C 180,E1 -13897.322,E2 -13897.322} C_VEL
LIN {X 0,Y 347.728,Z 340.792,A -85,B 0,C 180,E1 -13900.298,E2 -13900.298} C_VEL
LIN {X 0,Y 347.72,Z 340.797,A -85,B 0,C 180,E1 -13903.409,E2 -13903.409} C_VEL
LIN {X 0,Y 347.723,Z 340.795,A -85,B 0,C 180,E1 -13906.688,E2 -13906.688} C_VEL
LIN {X 0,Y 347.746,Z 340.793,A -85,B 0,C 180,E1 -13910.174,E2 -13910.174} C_VEL
LIN {X 0,Y 347.804,Z 340.926,A -85,B 0,C 180,E1 -13912.393,E2 -13912.393} C_VEL
LIN {X 0,Y 349.906,Z 349.037,A -85,B 0,C 180,E1 -13914.856,E2 -13914.856} C_VEL
LIN {X 0,Y 360.996,Z 372.591,A -85,B 0,C 180,E1 -13916.471,E2 -13916.471} C_VEL
LIN {X 0,Y 364.316,Z 380.84,A -85,B 0,C 180,E1 -13916.956,E2 -13916.956} C_VEL
LIN {X 0,Y 364.559,Z 383.785,A -85,B 0,C 180,E1 -13917.043,E2 -13917.043} C_VEL
LIN {X 0,Y 361.905,Z 484.953,A -85,B 0,C 180,E1 -13919.077,E2 -13919.077} C_VEL
LIN {X 0,Y 361.11,Z 499.763,A -85,B 0,C 180,E1 -13919.602,E2 -13919.602} C_VEL
LIN {X 0,Y 360.023,Z 513.36,A -85,B 0,C 180,E1 -13920.308,E2 -13920.308} C_VEL
LIN {X 0,Y 358.519,Z 527.496,A -85,B 0,C 180,E1 -13921.298,E2 -13921.298} C_VEL
LIN {X 0,Y 356.925,Z 540.055,A -85,B 0,C 180,E1 -13922.435,E2 -13922.435} C_VEL
LIN {X 0,Y 355.154,Z 551.534,A -85,B 0,C 180,E1 -13923.72,E2 -13923.72} C_VEL
LIN {X 0,Y 353.382,Z 563.005,A -85,B 0,C 180,E1 -13925.315,E2 -13925.315} C_VEL
LIN {X 0,Y 352.039,Z 571.924,A -85,B 0,C 180,E1 -13926.834,E2 -13926.834} C_VEL
LIN {X 0,Y 350.549,Z 580.327,A -85,B 0,C 180,E1 -13928.539,E2 -13928.539} C_VEL
LIN {X 0,Y 349.155,Z 588.609,A -85,B 0,C 180,E1 -13930.603,E2 -13930.603} C_VEL
LIN {X 0,Y 348.196,Z 594.378,A -85,B 0,C 180,E1 -13932.377,E2 -13932.377} C_VEL
LIN {X 0,Y 347.427,Z 599.075,A -85,B 0,C 180,E1 -13934.152,E2 -13934.152} C_VEL
LIN {X 0,Y 346.775,Z 604.075,A -85,B 0,C 180,E1 -13936.61,E2 -13936.61} C_VEL
LIN {X 0,Y 346.407,Z 606.525,A -85,B 0,C 180,E1 -13938.295,E2 -13938.295} C_VEL
LIN {X 0,Y 346.13,Z 608.775,A -85,B 0,C 180,E1 -13940.652,E2 -13940.652} C_VEL
LIN {X 0,Y 346.13,Z 609.671,A -85,B 0,C 180,E1 -13943.003,E2 -13943.003} C_VEL
LIN {X 0,Y 346.204,Z 609.622,A -85,B 0,C 180,E1 -13944.175,E2 -13944.175} C_VEL
LIN {X 0,Y 346.158,Z 608.541,A -85,B 0,C 180,E1 -13946.508,E2 -13946.508} C_VEL
LIN {X 0,Y 346.268,Z 606.13,A -85,B 0,C 180,E1 -13948.837,E2 -13948.837} C_VEL
LIN {X 0,Y 346.542,Z 602.331,A -85,B 0,C 180,E1 -13951.162,E2 -13951.162} C_VEL
LIN {X 0,Y 347.02,Z 596.986,A -85,B 0,C 180,E1 -13953.483,E2 -13953.483} C_VEL
LIN {X 0,Y 347.606,Z 591.891,A -85,B 0,C 180,E1 -13955.22,E2 -13955.22} C_VEL
LIN {X 0,Y 348.671,Z 584.581,A -85,B 0,C 180,E1 -13957.237,E2 -13957.237} C_VEL
LIN {X 0,Y 349.585,Z 576.947,A -85,B 0,C 180,E1 -13958.963,E2 -13958.963} C_VEL
LIN {X 0,Y 350.758,Z 567.968,A -85,B 0,C 180,E1 -13960.648,E2 -13960.648} C_VEL
LIN {X 0,Y 352.077,Z 557.669,A -85,B 0,C 180,E1 -13962.245,E2 -13962.245} C_VEL
LIN {X 0,Y 353.539,Z 546.521,A -85,B 0,C 180,E1 -13963.654,E2 -13963.654} C_VEL
LIN {X 0,Y 354.84,Z 534.228,A -85,B 0,C 180,E1 -13964.92,E2 -13964.92} C_VEL
LIN {X 0,Y 356.004,Z 522.395,A -85,B 0,C 180,E1 -13965.897,E2 -13965.897} C_VEL
LIN {X 0,Y 357.09,Z 509.457,A -85,B 0,C 180,E1 -13966.728,E2 -13966.728} C_VEL
LIN {X 0,Y 358.013,Z 495.528,A -85,B 0,C 180,E1 -13967.382,E2 -13967.382} C_VEL
LIN {X 0,Y 358.56,Z 480.984,A -85,B 0,C 180,E1 -13967.833,E2 -13967.833} C_VEL
LIN {X 0,Y 359.123,Z 451.241,A -85,B 0,C 180,E1 -13968.438,E2 -13968.438} C_VEL
LIN {X 0,Y 358.619,Z 445.436,A -85,B 0,C 180,E1 -13968.594,E2 -13968.594} C_VEL
LIN {X 0,Y 353.706,Z 426.767,A -85,B 0,C 180,E1 -13969.328,E2 -13969.328} C_VEL
LIN {X 0,Y 353.248,Z 420.962,A -85,B 0,C 180,E1 -13969.486,E2 -13969.486} C_VEL
LIN {X 0,Y 354.009,Z 380.708,A -85,B 0,C 180,E1 -13970.308,E2 -13970.308} C_VEL
LIN {X 0,Y 352.6,Z 374.54,A -85,B 0,C 180,E1 -13970.546,E2 -13970.546} C_VEL
LIN {X 0,Y 344.791,Z 354.667,A -85,B 0,C 180,E1 -13971.584,E2 -13971.584} C_VEL
LIN {X 0,Y 342.301,Z 348.64,A -85,B 0,C 180,E1 -13971.951,E2 -13971.951} C_VEL
LIN {X 0,Y 340.746,Z 341.667,A -85,B 0,C 180,E1 -13973.957,E2 -13973.957} C_VEL
LIN {X 0,Y 340.778,Z 341.664,A -85,B 0,C 180,E1 -13977.524,E2 -13977.524} C_VEL
LIN {X 0,Y 340.699,Z 341.671,A -85,B 0,C 180,E1 -13981.044,E2 -13981.044} C_VEL
LIN {X 0,Y 340.719,Z 341.661,A -85,B 0,C 180,E1 -13985.278,E2 -13985.278} C_VEL
LIN {X 0,Y 340.711,Z 341.667,A -85,B 0,C 180,E1 -13988.385,E2 -13988.385} C_VEL
LIN {X 0,Y 340.697,Z 341.669,A -85,B 0,C 180,E1 -13992.044,E2 -13992.044} C_VEL
LIN {X 0,Y 340.649,Z 341.676,A -85,B 0,C 180,E1 -13996.226,E2 -13996.226} C_VEL
LIN {X 0,Y 340.684,Z 341.673,A -85,B 0,C 180,E1 -13999.752,E2 -13999.752} C_VEL
LIN {X 0,Y 340.7,Z 341.668,A -85,B 0,C 180,E1 -14003.257,E2 -14003.257} C_VEL
LIN {X 0,Y 340.687,Z 341.666,A -85,B 0,C 180,E1 -14006.152,E2 -14006.152} C_VEL
LIN {X 0,Y 340.735,Z 341.664,A -85,B 0,C 180,E1 -14010.328,E2 -14010.328} C_VEL
LIN {X 0,Y 340.773,Z 341.648,A -85,B 0,C 180,E1 -14013.017,E2 -14013.017} C_VEL
LIN {X 0,Y 340.744,Z 341.664,A -85,B 0,C 180,E1 -14015.637,E2 -14015.637} C_VEL
LIN {X 0,Y 340.712,Z 341.651,A -85,B 0,C 180,E1 -14019.471,E2 -14019.471} C_VEL
LIN {X 0,Y 340.784,Z 341.655,A -85,B 0,C 180,E1 -14021.98,E2 -14021.98} C_VEL
LIN {X 0,Y 340.844,Z 341.643,A -85,B 0,C 180,E1 -14025.716,E2 -14025.716} C_VEL
LIN {X 0,Y 340.837,Z 341.649,A -85,B 0,C 180,E1 -14029.305,E2 -14029.305} C_VEL
LIN {X 0,Y 341.031,Z 341.624,A -85,B 0,C 180,E1 -14032.897,E2 -14032.897} C_VEL
LIN {X 0,Y 341.118,Z 341.611,A -85,B 0,C 180,E1 -14037.638,E2 -14037.638} C_VEL
LIN {X 0,Y 341.096,Z 341.616,A -85,B 0,C 180,E1 -14041.18,E2 -14041.18} C_VEL
LIN {X 0,Y 340.824,Z 341.643,A -85,B 0,C 180,E1 -14043.546,E2 -14043.546} C_VEL
LIN {X 0,Y 340.999,Z 341.632,A -85,B 0,C 180,E1 -14045.914,E2 -14045.914} C_VEL
LIN {X 0,Y 340.954,Z 341.632,A -85,B 0,C 180,E1 -14048.356,E2 -14048.356} C_VEL
LIN {X 0,Y 340.837,Z 341.652,A -85,B 0,C 180,E1 -14051.899,E2 -14051.899} C_VEL
LIN {X 0,Y 340.807,Z 341.646,A -85,B 0,C 180,E1 -14055.55,E2 -14055.55} C_VEL
LIN {X 0,Y 340.747,Z 341.661,A -85,B 0,C 180,E1 -14059.269,E2 -14059.269} C_VEL
LIN {X 0,Y 340.704,Z 341.666,A -85,B 0,C 180,E1 -14063.074,E2 -14063.074} C_VEL
LIN {X 0,Y 340.715,Z 341.662,A -85,B 0,C 180,E1 -14065.669,E2 -14065.669} C_VEL
LIN {X 0,Y 340.696,Z 341.668,A -85,B 0,C 180,E1 -14069.675,E2 -14069.675} C_VEL
LIN {X 0,Y 340.678,Z 341.673,A -85,B 0,C 180,E1 -14072.436,E2 -14072.436} C_VEL
LIN {X 0,Y 340.71,Z 341.667,A -85,B 0,C 180,E1 -14075.28,E2 -14075.28} C_VEL
LIN {X 0,Y 340.703,Z 341.67,A -85,B 0,C 180,E1 -14078.387,E2 -14078.387} C_VEL
LIN {X 0,Y 340.692,Z 341.661,A -85,B 0,C 180,E1 -14082.046,E2 -14082.046} C_VEL
LIN {X 0,Y 340.646,Z 341.677,A -85,B 0,C 180,E1 -14086.228,E2 -14086.228} C_VEL
LIN {X 0,Y 340.683,Z 341.676,A -85,B 0,C 180,E1 -14089.754,E2 -14089.754} C_VEL
LIN {X 0,Y 340.7,Z 341.677,A -85,B 0,C 180,E1 -14093.259,E2 -14093.259} C_VEL
LIN {X 0,Y 340.747,Z 341.818,A -85,B 0,C 180,E1 -14096.307,E2 -14096.307} C_VEL
LIN {X 0,Y 343.635,Z 354.013,A -85,B 0,C 180,E1 -14099.504,E2 -14099.504} C_VEL
LIN {X 0,Y 346.074,Z 365.797,A -85,B 0,C 180,E1 -14102.405,E2 -14102.405} C_VEL
LIN {X 0,Y 347.704,Z 371.15,A -85,B 0,C 180,E1 -14102.65,E2 -14102.65} C_VEL
LIN {X 0,Y 352.172,Z 397.576,A -85,B 0,C 180,E1 -14103.565,E2 -14103.565} C_VEL
LIN {X 0,Y 353.669,Z 406.984,A -85,B 0,C 180,E1 -14103.878,E2 -14103.878} C_VEL
LIN {X 0,Y 351.502,Z 503.292,A -85,B 0,C 180,E1 -14105.843,E2 -14105.843} C_VEL
LIN {X 0,Y 350.734,Z 517.399,A -85,B 0,C 180,E1 -14106.336,E2 -14106.336} C_VEL
LIN {X 0,Y 349.622,Z 531.696,A -85,B 0,C 180,E1 -14107.079,E2 -14107.079} C_VEL
LIN {X 0,Y 348.291,Z 545.521,A -85,B 0,C 180,E1 -14108.057,E2 -14108.057} C_VEL
LIN {X 0,Y 346.823,Z 558.383,A -85,B 0,C 180,E1 -14109.231,E2 -14109.231} C_VEL
LIN {X 0,Y 345.189,Z 571.053,A -85,B 0,C 180,E1 -14110.68,E2 -14110.68} C_VEL
LIN {X 0,Y 343.817,Z 581.406,A -85,B 0,C 180,E1 -14112.145,E2 -14112.145} C_VEL
LIN {X 0,Y 342.403,Z 591.682,A -85,B 0,C 180,E1 -14113.914,E2 -14113.914} C_VEL
LIN {X 0,Y 341.437,Z 600.203,A -85,B 0,C 180,E1 -14115.7,E2 -14115.7} C_VEL
LIN {X 0,Y 340.438,Z 608.325,A -85,B 0,C 180,E1 -14117.784,E2 -14117.784} C_VEL
LIN {X 0,Y 339.693,Z 614.861,A -85,B 0,C 180,E1 -14119.872,E2 -14119.872} C_VEL
LIN {X 0,Y 339.295,Z 620.655,A -85,B 0,C 180,E1 -14122.263,E2 -14122.263} C_VEL
LIN {X 0,Y 339.149,Z 624.006,A -85,B 0,C 180,E1 -14124.085,E2 -14124.085} C_VEL
LIN {X 0,Y 339.065,Z 627.04,A -85,B 0,C 180,E1 -14126.435,E2 -14126.435} C_VEL
LIN {X 0,Y 339.021,Z 628.736,A -85,B 0,C 180,E1 -14128.812,E2 -14128.812} C_VEL
LIN {X 0,Y 339.066,Z 629.081,A -85,B 0,C 180,E1 -14130,E2 -14130} C_VEL
LIN {X 0,Y 338.994,Z 628.763,A -85,B 0,C 180,E1 -14132.376,E2 -14132.376} C_VEL
LIN {X 0,Y 339.05,Z 627.114,A -85,B 0,C 180,E1 -14134.756,E2 -14134.756} C_VEL
LIN {X 0,Y 339.259,Z 624.1,A -85,B 0,C 180,E1 -14137.14,E2 -14137.14} C_VEL
LIN {X 0,Y 339.679,Z 619.643,A -85,B 0,C 180,E1 -14139.527,E2 -14139.527} C_VEL
LIN {X 0,Y 340.45,Z 613.601,A -85,B 0,C 180,E1 -14141.913,E2 -14141.913} C_VEL
LIN {X 0,Y 341.518,Z 606.83,A -85,B 0,C 180,E1 -14143.992,E2 -14143.992} C_VEL
LIN {X 0,Y 342.86,Z 598.436,A -85,B 0,C 180,E1 -14146.064,E2 -14146.064} C_VEL
LIN {X 0,Y 344.401,Z 589.708,A -85,B 0,C 180,E1 -14147.824,E2 -14147.824} C_VEL
LIN {X 0,Y 346.249,Z 579.154,A -85,B 0,C 180,E1 -14149.566,E2 -14149.566} C_VEL
LIN {X 0,Y 348.234,Z 567.355,A -85,B 0,C 180,E1 -14151.146,E2 -14151.146} C_VEL
LIN {X 0,Y 350.015,Z 555.53,A -85,B 0,C 180,E1 -14152.426,E2 -14152.426} C_VEL
LIN {X 0,Y 351.705,Z 542.485,A -85,B 0,C 180,E1 -14153.556,E2 -14153.556} C_VEL
LIN {X 0,Y 353.254,Z 528.746,A -85,B 0,C 180,E1 -14154.46,E2 -14154.46} C_VEL
LIN {X 0,Y 354.593,Z 514.198,A -85,B 0,C 180,E1 -14155.143,E2 -14155.143} C_VEL
LIN {X 0,Y 355.381,Z 499.758,A -85,B 0,C 180,E1 -14155.593,E2 -14155.593} C_VEL
LIN {X 0,Y 357.757,Z 407.45,A -85,B 0,C 180,E1 -14157.476,E2 -14157.476} C_VEL
LIN {X 0,Y 352.974,Z 382.542,A -85,B 0,C 180,E1 -14158.494,E2 -14158.494} C_VEL
LIN {X 0,Y 351.381,Z 376.182,A -85,B 0,C 180,E1 -14158.796,E2 -14158.796} C_VEL
LIN {X 0,Y 346.619,Z 365.268,A -85,B 0,C 180,E1 -14159.534,E2 -14159.534} C_VEL
LIN {X 0,Y 343.85,Z 353.628,A -85,B 0,C 180,E1 -14162.714,E2 -14162.714} C_VEL
LIN {X 0,Y 341.28,Z 343.757,A -85,B 0,C 180,E1 -14165.573,E2 -14165.573} C_VEL
LIN {X 0,Y 340.719,Z 341.664,A -85,B 0,C 180,E1 -14166.221,E2 -14166.221} C_VEL
LIN {X 0,Y 340.694,Z 341.658,A -85,B 0,C 180,E1 -14169.752,E2 -14169.752} C_VEL
LIN {X 0,Y 340.67,Z 341.666,A -85,B 0,C 180,E1 -14172.904,E2 -14172.904} C_VEL
LIN {X 0,Y 340.67,Z 341.669,A -85,B 0,C 180,E1 -14177.095,E2 -14177.095} C_VEL
LIN {X 0,Y 340.692,Z 341.67,A -85,B 0,C 180,E1 -14180.247,E2 -14180.247} C_VEL
LIN {X 0,Y 340.703,Z 341.67,A -85,B 0,C 180,E1 -14183.559,E2 -14183.559} C_VEL
LIN {X 0,Y 340.685,Z 341.672,A -85,B 0,C 180,E1 -14186.153,E2 -14186.153} C_VEL
LIN {X 0,Y 340.713,Z 341.642,A -85,B 0,C 180,E1 -14190.034,E2 -14190.034} C_VEL
LIN {X 0,Y 340.712,Z 341.666,A -85,B 0,C 180,E1 -14193.012,E2 -14193.012} C_VEL
LIN {X 0,Y 340.732,Z 341.66,A -85,B 0,C 180,E1 -14195.637,E2 -14195.637} C_VEL
LIN {X 0,Y 340.719,Z 341.662,A -85,B 0,C 180,E1 -14199.473,E2 -14199.473} C_VEL
LIN {X 0,Y 340.783,Z 341.66,A -85,B 0,C 180,E1 -14201.98,E2 -14201.98} C_VEL
LIN {X 0,Y 340.843,Z 341.655,A -85,B 0,C 180,E1 -14205.716,E2 -14205.716} C_VEL
LIN {X 0,Y 340.831,Z 341.648,A -85,B 0,C 180,E1 -14209.305,E2 -14209.305} C_VEL
LIN {X 0,Y 340.991,Z 341.625,A -85,B 0,C 180,E1 -14212.897,E2 -14212.897} C_VEL
LIN {X 0,Y 340.803,Z 341.659,A -85,B 0,C 180,E1 -14215.269,E2 -14215.269} C_VEL
LIN {X 0,Y 341.115,Z 341.61,A -85,B 0,C 180,E1 -14217.639,E2 -14217.639} C_VEL
LIN {X 0,Y 341.077,Z 341.623,A -85,B 0,C 180,E1 -14221.181,E2 -14221.181} C_VEL
LIN {X 0,Y 341.122,Z 341.609,A -85,B 0,C 180,E1 -14222.362,E2 -14222.362} C_VEL
LIN {X 0,Y 341.01,Z 341.625,A -85,B 0,C 180,E1 -14227.104,E2 -14227.104} C_VEL
LIN {X 0,Y 340.837,Z 341.654,A -85,B 0,C 180,E1 -14230.695,E2 -14230.695} C_VEL
LIN {X 0,Y 340.855,Z 341.65,A -85,B 0,C 180,E1 -14234.326,E2 -14234.326} C_VEL
LIN {X 0,Y 340.778,Z 341.66,A -85,B 0,C 180,E1 -14238.441,E2 -14238.441} C_VEL
LIN {X 0,Y 340.711,Z 341.667,A -85,B 0,C 180,E1 -14241.843,E2 -14241.843} C_VEL
LIN {X 0,Y 340.765,Z 341.661,A -85,B 0,C 180,E1 -14245.666,E2 -14245.666} C_VEL
LIN {X 0,Y 340.722,Z 341.662,A -85,B 0,C 180,E1 -14248.322,E2 -14248.322} C_VEL
LIN {X 0,Y 340.692,Z 341.666,A -85,B 0,C 180,E1 -14251.046,E2 -14251.046} C_VEL
LIN {X 0,Y 340.713,Z 341.668,A -85,B 0,C 180,E1 -14255.28,E2 -14255.28} C_VEL
LIN {X 0,Y 340.705,Z 341.668,A -85,B 0,C 180,E1 -14258.387,E2 -14258.387} C_VEL
LIN {X 0,Y 340.696,Z 341.67,A -85,B 0,C 180,E1 -14262.047,E2 -14262.047} C_VEL
LIN {X 0,Y 340.65,Z 341.679,A -85,B 0,C 180,E1 -14266.228,E2 -14266.228} C_VEL
LIN {X 0,Y 340.688,Z 341.675,A -85,B 0,C 180,E1 -14269.754,E2 -14269.754} C_VEL
LIN {X 0,Y 340.735,Z 341.798,A -85,B 0,C 180,E1 -14271.774,E2 -14271.774} C_VEL
LIN {X 0,Y 342.674,Z 349.15,A -85,B 0,C 180,E1 -14274.107,E2 -14274.107} C_VEL
LIN {X 0,Y 353.143,Z 370.974,A -85,B 0,C 180,E1 -14275.692,E2 -14275.692} C_VEL
LIN {X 0,Y 358.375,Z 383.177,A -85,B 0,C 180,E1 -14276.468,E2 -14276.468} C_VEL
LIN {X 0,Y 355.604,Z 485.336,A -85,B 0,C 180,E1 -14278.558,E2 -14278.558} C_VEL
LIN {X 0,Y 354.809,Z 499.92,A -85,B 0,C 180,E1 -14279.086,E2 -14279.086} C_VEL
LIN {X 0,Y 353.666,Z 513.525,A -85,B 0,C 180,E1 -14279.802,E2 -14279.802} C_VEL
LIN {X 0,Y 352.2,Z 526.771,A -85,B 0,C 180,E1 -14280.733,E2 -14280.733} C_VEL
LIN {X 0,Y 350.586,Z 539.503,A -85,B 0,C 180,E1 -14281.891,E2 -14281.891} C_VEL
LIN {X 0,Y 348.683,Z 551.118,A -85,B 0,C 180,E1 -14283.194,E2 -14283.194} C_VEL
LIN {X 0,Y 347.143,Z 560.738,A -85,B 0,C 180,E1 -14284.52,E2 -14284.52} C_VEL
LIN {X 0,Y 345.389,Z 571.39,A -85,B 0,C 180,E1 -14286.302,E2 -14286.302} C_VEL
LIN {X 0,Y 343.829,Z 580.173,A -85,B 0,C 180,E1 -14288.098,E2 -14288.098} C_VEL
LIN {X 0,Y 342.313,Z 588.541,A -85,B 0,C 180,E1 -14290.199,E2 -14290.199} C_VEL
LIN {X 0,Y 341.31,Z 594.341,A -85,B 0,C 180,E1 -14292.009,E2 -14292.009} C_VEL
LIN {X 0,Y 340.48,Z 599.089,A -85,B 0,C 180,E1 -14293.82,E2 -14293.82} C_VEL
LIN {X 0,Y 339.926,Z 602.916,A -85,B 0,C 180,E1 -14295.635,E2 -14295.635} C_VEL
LIN {X 0,Y 339.355,Z 606.632,A -85,B 0,C 180,E1 -14298.048,E2 -14298.048} C_VEL
LIN {X 0,Y 339.063,Z 608.925,A -85,B 0,C 180,E1 -14300.455,E2 -14300.455} C_VEL
LIN {X 0,Y 339.038,Z 609.863,A -85,B 0,C 180,E1 -14302.855,E2 -14302.855} C_VEL
LIN {X 0,Y 339.115,Z 609.821,A -85,B 0,C 180,E1 -14304.149,E2 -14304.149} C_VEL
LIN {X 0,Y 339.081,Z 608.795,A -85,B 0,C 180,E1 -14306.435,E2 -14306.435} C_VEL
LIN {X 0,Y 339.166,Z 606.426,A -85,B 0,C 180,E1 -14308.813,E2 -14308.813} C_VEL
LIN {X 0,Y 339.479,Z 602.672,A -85,B 0,C 180,E1 -14311.186,E2 -14311.186} C_VEL
LIN {X 0,Y 339.973,Z 597.396,A -85,B 0,C 180,E1 -14313.555,E2 -14313.555} C_VEL
LIN {X 0,Y 340.576,Z 592.327,A -85,B 0,C 180,E1 -14315.328,E2 -14315.328} C_VEL
LIN {X 0,Y 341.665,Z 585.078,A -85,B 0,C 180,E1 -14317.386,E2 -14317.386} C_VEL
LIN {X 0,Y 342.607,Z 577.5,A -85,B 0,C 180,E1 -14319.147,E2 -14319.147} C_VEL
LIN {X 0,Y 343.929,Z 567.948,A -85,B 0,C 180,E1 -14320.98,E2 -14320.98} C_VEL
LIN {X 0,Y 345.301,Z 557.378,A -85,B 0,C 180,E1 -14322.638,E2 -14322.638} C_VEL
LIN {X 0,Y 346.822,Z 546.113,A -85,B 0,C 180,E1 -14324.073,E2 -14324.073} C_VEL
LIN {X 0,Y 348.202,Z 533.677,A -85,B 0,C 180,E1 -14325.361,E2 -14325.361} C_VEL
LIN {X 0,Y 349.439,Z 521.646,A -85,B 0,C 180,E1 -14326.353,E2 -14326.353} C_VEL
LIN {X 0,Y 350.587,Z 508.409,A -85,B 0,C 180,E1 -14327.198,E2 -14327.198} C_VEL
LIN {X 0,Y 351.512,Z 493.982,A -85,B 0,C 180,E1 -14327.865,E2 -14327.865} C_VEL
LIN {X 0,Y 352.027,Z 479.809,A -85,B 0,C 180,E1 -14328.289,E2 -14328.289} C_VEL
LIN {X 0,Y 353.248,Z 420.962,A -85,B 0,C 180,E1 -14329.486,E2 -14329.486} C_VEL
LIN {X 0,Y 352.798,Z 415.157,A -85,B 0,C 180,E1 -14329.644,E2 -14329.644} C_VEL
LIN {X 0,Y 347.978,Z 396.485,A -85,B 0,C 180,E1 -14330.403,E2 -14330.403} C_VEL
LIN {X 0,Y 347.479,Z 390.681,A -85,B 0,C 180,E1 -14330.57,E2 -14330.57} C_VEL
LIN {X 0,Y 347.494,Z 381.727,A -85,B 0,C 180,E1 -14330.768,E2 -14330.768} C_VEL
LIN {X 0,Y 346.241,Z 376.589,A -85,B 0,C 180,E1 -14330.978,E2 -14330.978} C_VEL
LIN {X 0,Y 339.094,Z 358.238,A -85,B 0,C 180,E1 -14331.96,E2 -14331.96} C_VEL
LIN {X 0,Y 335.137,Z 348.85,A -85,B 0,C 180,E1 -14332.54,E2 -14332.54} C_VEL
LIN {X 0,Y 333.722,Z 342.542,A -85,B 0,C 180,E1 -14334.411,E2 -14334.411} C_VEL
LIN {X 0,Y 333.718,Z 342.541,A -85,B 0,C 180,E1 -14337.808,E2 -14337.808} C_VEL
LIN {X 0,Y 333.691,Z 342.544,A -85,B 0,C 180,E1 -14340.362,E2 -14340.362} C_VEL
LIN {X 0,Y 333.674,Z 342.543,A -85,B 0,C 180,E1 -14344.657,E2 -14344.657} C_VEL
LIN {X 0,Y 333.654,Z 342.551,A -85,B 0,C 180,E1 -14347.65,E2 -14347.65} C_VEL
LIN {X 0,Y 333.645,Z 342.531,A -85,B 0,C 180,E1 -14350.766,E2 -14350.766} C_VEL
LIN {X 0,Y 333.591,Z 342.552,A -85,B 0,C 180,E1 -14354.249,E2 -14354.249} C_VEL
LIN {X 0,Y 333.638,Z 342.546,A -85,B 0,C 180,E1 -14357.617,E2 -14357.617} C_VEL
LIN {X 0,Y 333.648,Z 342.548,A -85,B 0,C 180,E1 -14361.201,E2 -14361.201} C_VEL
LIN {X 0,Y 333.671,Z 342.546,A -85,B 0,C 180,E1 -14363.86,E2 -14363.86} C_VEL
LIN {X 0,Y 333.638,Z 342.546,A -85,B 0,C 180,E1 -14367.412,E2 -14367.412} C_VEL
LIN {X 0,Y 333.681,Z 342.538,A -85,B 0,C 180,E1 -14371.025,E2 -14371.025} C_VEL
LIN {X 0,Y 333.712,Z 342.535,A -85,B 0,C 180,E1 -14373.751,E2 -14373.751} C_VEL
LIN {X 0,Y 333.647,Z 342.542,A -85,B 0,C 180,E1 -14377.718,E2 -14377.718} C_VEL
LIN {X 0,Y 333.732,Z 342.534,A -85,B 0,C 180,E1 -14381.585,E2 -14381.585} C_VEL
LIN {X 0,Y 333.8,Z 342.52,A -85,B 0,C 180,E1 -14385.576,E2 -14385.576} C_VEL
LIN {X 0,Y 333.807,Z 342.52,A -85,B 0,C 180,E1 -14389.077,E2 -14389.077} C_VEL
LIN {X 0,Y 333.979,Z 342.504,A -85,B 0,C 180,E1 -14392.746,E2 -14392.746} C_VEL
LIN {X 0,Y 333.779,Z 342.51,A -85,B 0,C 180,E1 -14395.168,E2 -14395.168} C_VEL
LIN {X 0,Y 334.059,Z 342.491,A -85,B 0,C 180,E1 -14397.588,E2 -14397.588} C_VEL
LIN {X 0,Y 334.064,Z 342.492,A -85,B 0,C 180,E1 -14401.205,E2 -14401.205} C_VEL
LIN {X 0,Y 333.773,Z 342.521,A -85,B 0,C 180,E1 -14403.621,E2 -14403.621} C_VEL
LIN {X 0,Y 333.974,Z 342.508,A -85,B 0,C 180,E1 -14406.039,E2 -14406.039} C_VEL
LIN {X 0,Y 333.903,Z 342.508,A -85,B 0,C 180,E1 -14408.472,E2 -14408.472} C_VEL
LIN {X 0,Y 333.779,Z 342.533,A -85,B 0,C 180,E1 -14412.155,E2 -14412.155} C_VEL
LIN {X 0,Y 333.799,Z 342.521,A -85,B 0,C 180,E1 -14414.634,E2 -14414.634} C_VEL
LIN {X 0,Y 333.743,Z 342.536,A -85,B 0,C 180,E1 -14418.632,E2 -14418.632} C_VEL
LIN {X 0,Y 333.645,Z 342.543,A -85,B 0,C 180,E1 -14422.281,E2 -14422.281} C_VEL
LIN {X 0,Y 333.683,Z 342.538,A -85,B 0,C 180,E1 -14425.091,E2 -14425.091} C_VEL
LIN {X 0,Y 333.645,Z 342.546,A -85,B 0,C 180,E1 -14428.978,E2 -14428.978} C_VEL
LIN {X 0,Y 333.636,Z 342.549,A -85,B 0,C 180,E1 -14432.587,E2 -14432.587} C_VEL
LIN {X 0,Y 333.669,Z 342.547,A -85,B 0,C 180,E1 -14436.14,E2 -14436.14} C_VEL
LIN {X 0,Y 333.64,Z 342.55,A -85,B 0,C 180,E1 -14439.193,E2 -14439.193} C_VEL
LIN {X 0,Y 333.626,Z 342.545,A -85,B 0,C 180,E1 -14442.501,E2 -14442.501} C_VEL
LIN {X 0,Y 333.591,Z 342.558,A -85,B 0,C 180,E1 -14445.956,E2 -14445.956} C_VEL
LIN {X 0,Y 333.642,Z 342.553,A -85,B 0,C 180,E1 -14449.316,E2 -14449.316} C_VEL
LIN {X 0,Y 333.661,Z 342.553,A -85,B 0,C 180,E1 -14453.169,E2 -14453.169} C_VEL
LIN {X 0,Y 333.7,Z 342.722,A -85,B 0,C 180,E1 -14455.848,E2 -14455.848} C_VEL
LIN {X 0,Y 336.412,Z 354.149,A -85,B 0,C 180,E1 -14458.929,E2 -14458.929} C_VEL
LIN {X 0,Y 338.897,Z 365.664,A -85,B 0,C 180,E1 -14461.833,E2 -14461.833} C_VEL
LIN {X 0,Y 341.303,Z 372.459,A -85,B 0,C 180,E1 -14462.182,E2 -14462.182} C_VEL
LIN {X 0,Y 346.17,Z 401.405,A -85,B 0,C 180,E1 -14463.209,E2 -14463.209} C_VEL
LIN {X 0,Y 347.169,Z 407.934,A -85,B 0,C 180,E1 -14463.429,E2 -14463.429} C_VEL
LIN {X 0,Y 344.954,Z 502.687,A -85,B 0,C 180,E1 -14465.394,E2 -14465.394} C_VEL
LIN {X 0,Y 344.161,Z 516.976,A -85,B 0,C 180,E1 -14465.896,E2 -14465.896} C_VEL
LIN {X 0,Y 343.044,Z 530.76,A -85,B 0,C 180,E1 -14466.614,E2 -14466.614} C_VEL
LIN {X 0,Y 341.852,Z 543.167,A -85,B 0,C 180,E1 -14467.48,E2 -14467.48} C_VEL
LIN {X 0,Y 340.355,Z 556.285,A -85,B 0,C 180,E1 -14468.658,E2 -14468.658} C_VEL
LIN {X 0,Y 338.769,Z 568.106,A -85,B 0,C 180,E1 -14469.983,E2 -14469.983} C_VEL
LIN {X 0,Y 337.257,Z 578.919,A -85,B 0,C 180,E1 -14471.471,E2 -14471.471} C_VEL
LIN {X 0,Y 335.742,Z 589.622,A -85,B 0,C 180,E1 -14473.273,E2 -14473.273} C_VEL
LIN {X 0,Y 334.642,Z 598.188,A -85,B 0,C 180,E1 -14475.032,E2 -14475.032} C_VEL
LIN {X 0,Y 333.707,Z 605.79,A -85,B 0,C 180,E1 -14476.915,E2 -14476.915} C_VEL
LIN {X 0,Y 332.812,Z 612.8,A -85,B 0,C 180,E1 -14479.044,E2 -14479.044} C_VEL
LIN {X 0,Y 332.389,Z 617.651,A -85,B 0,C 180,E1 -14480.876,E2 -14480.876} C_VEL
LIN {X 0,Y 332.103,Z 622.66,A -85,B 0,C 180,E1 -14483.316,E2 -14483.316} C_VEL
LIN {X 0,Y 331.98,Z 625.417,A -85,B 0,C 180,E1 -14485.143,E2 -14485.143} C_VEL
LIN {X 0,Y 331.99,Z 626.795,A -85,B 0,C 180,E1 -14486.359,E2 -14486.359} C_VEL
LIN {X 0,Y 331.926,Z 628.516,A -85,B 0,C 180,E1 -14488.787,E2 -14488.787} C_VEL
LIN {X 0,Y 331.969,Z 628.873,A -85,B 0,C 180,E1 -14490,E2 -14490} C_VEL
LIN {X 0,Y 331.911,Z 628.58,A -85,B 0,C 180,E1 -14492.427,E2 -14492.427} C_VEL
LIN {X 0,Y 331.959,Z 626.956,A -85,B 0,C 180,E1 -14494.858,E2 -14494.858} C_VEL
LIN {X 0,Y 332.182,Z 623.968,A -85,B 0,C 180,E1 -14497.293,E2 -14497.293} C_VEL
LIN {X 0,Y 332.633,Z 619.538,A -85,B 0,C 180,E1 -14499.731,E2 -14499.731} C_VEL
LIN {X 0,Y 333.485,Z 613.538,A -85,B 0,C 180,E1 -14502.166,E2 -14502.166} C_VEL
LIN {X 0,Y 334.586,Z 606.805,A -85,B 0,C 180,E1 -14504.288,E2 -14504.288} C_VEL
LIN {X 0,Y 335.988,Z 598.451,A -85,B 0,C 180,E1 -14506.402,E2 -14506.402} C_VEL
LIN {X 0,Y 337.625,Z 589.768,A -85,B 0,C 180,E1 -14508.194,E2 -14508.194} C_VEL
LIN {X 0,Y 339.569,Z 579.266,A -85,B 0,C 180,E1 -14509.968,E2 -14509.968} C_VEL
LIN {X 0,Y 341.631,Z 567.532,A -85,B 0,C 180,E1 -14511.575,E2 -14511.575} C_VEL
LIN {X 0,Y 343.456,Z 555.791,A -85,B 0,C 180,E1 -14512.879,E2 -14512.879} C_VEL
LIN {X 0,Y 345.228,Z 542.855,A -85,B 0,C 180,E1 -14514.025,E2 -14514.025} C_VEL
LIN {X 0,Y 346.84,Z 529.356,A -85,B 0,C 180,E1 -14514.943,E2 -14514.943} C_VEL
LIN {X 0,Y 348.233,Z 515.179,A -85,B 0,C 180,E1 -14515.635,E2 -14515.635} C_VEL
LIN {X 0,Y 349.083,Z 501.492,A -85,B 0,C 180,E1 -14516.089,E2 -14516.089} C_VEL
LIN {X 0,Y 351.579,Z 408.491,A -85,B 0,C 180,E1 -14518.025,E2 -14518.025} C_VEL
LIN {X 0,Y 347.014,Z 384.497,A -85,B 0,C 180,E1 -14519.032,E2 -14519.032} C_VEL
LIN {X 0,Y 345.73,Z 379.306,A -85,B 0,C 180,E1 -14519.285,E2 -14519.285} C_VEL
LIN {X 0,Y 339.345,Z 364.903,A -85,B 0,C 180,E1 -14520.334,E2 -14520.334} C_VEL
LIN {X 0,Y 336.152,Z 351.748,A -85,B 0,C 180,E1 -14524.07,E2 -14524.07} C_VEL
LIN {X 0,Y 333.668,Z 342.535,A -85,B 0,C 180,E1 -14526.898,E2 -14526.898} C_VEL
LIN {X 0,Y 333.641,Z 342.533,A -85,B 0,C 180,E1 -14530.767,E2 -14530.767} C_VEL
LIN {X 0,Y 333.588,Z 342.554,A -85,B 0,C 180,E1 -14534.25,E2 -14534.25} C_VEL
LIN {X 0,Y 333.635,Z 342.545,A -85,B 0,C 180,E1 -14537.618,E2 -14537.618} C_VEL
LIN {X 0,Y 333.646,Z 342.549,A -85,B 0,C 180,E1 -14541.202,E2 -14541.202} C_VEL
LIN {X 0,Y 333.669,Z 342.548,A -85,B 0,C 180,E1 -14543.86,E2 -14543.86} C_VEL
LIN {X 0,Y 333.636,Z 342.55,A -85,B 0,C 180,E1 -14547.413,E2 -14547.413} C_VEL
LIN {X 0,Y 333.645,Z 342.527,A -85,B 0,C 180,E1 -14551.022,E2 -14551.022} C_VEL
LIN {X 0,Y 333.688,Z 342.538,A -85,B 0,C 180,E1 -14555.088,E2 -14555.088} C_VEL
LIN {X 0,Y 333.653,Z 342.543,A -85,B 0,C 180,E1 -14559.018,E2 -14559.018} C_VEL
LIN {X 0,Y 333.731,Z 342.54,A -85,B 0,C 180,E1 -14561.586,E2 -14561.586} C_VEL
LIN {X 0,Y 333.799,Z 342.53,A -85,B 0,C 180,E1 -14565.577,E2 -14565.577} C_VEL
LIN {X 0,Y 333.802,Z 342.521,A -85,B 0,C 180,E1 -14569.077,E2 -14569.077} C_VEL
LIN {X 0,Y 333.946,Z 342.503,A -85,B 0,C 180,E1 -14572.746,E2 -14572.746} C_VEL
LIN {X 0,Y 333.769,Z 342.534,A -85,B 0,C 180,E1 -14575.169,E2 -14575.169} C_VEL
LIN {X 0,Y 334.055,Z 342.489,A -85,B 0,C 180,E1 -14577.589,E2 -14577.589} C_VEL
LIN {X 0,Y 334.048,Z 342.498,A -85,B 0,C 180,E1 -14581.206,E2 -14581.206} C_VEL
LIN {X 0,Y 334.063,Z 342.488,A -85,B 0,C 180,E1 -14582.412,E2 -14582.412} C_VEL
LIN {X 0,Y 333.958,Z 342.503,A -85,B 0,C 180,E1 -14586.587,E2 -14586.587} C_VEL
LIN {X 0,Y 333.811,Z 342.529,A -85,B 0,C 180,E1 -14589.697,E2 -14589.697} C_VEL
LIN {X 0,Y 333.788,Z 342.53,A -85,B 0,C 180,E1 -14593.392,E2 -14593.392} C_VEL
LIN {X 0,Y 333.71,Z 342.536,A -85,B 0,C 180,E1 -14597.149,E2 -14597.149} C_VEL
LIN {X 0,Y 333.663,Z 342.543,A -85,B 0,C 180,E1 -14599.695,E2 -14599.695} C_VEL
LIN {X 0,Y 333.663,Z 342.544,A -85,B 0,C 180,E1 -14603.591,E2 -14603.591} C_VEL
LIN {X 0,Y 333.728,Z 342.539,A -85,B 0,C 180,E1 -14606.247,E2 -14606.247} C_VEL
LIN {X 0,Y 333.684,Z 342.543,A -85,B 0,C 180,E1 -14608.975,E2 -14608.975} C_VEL
LIN {X 0,Y 333.638,Z 342.549,A -85,B 0,C 180,E1 -14612.588,E2 -14612.588} C_VEL
LIN {X 0,Y 333.671,Z 342.546,A -85,B 0,C 180,E1 -14616.14,E2 -14616.14} C_VEL
LIN {X 0,Y 333.643,Z 342.547,A -85,B 0,C 180,E1 -14619.194,E2 -14619.194} C_VEL
LIN {X 0,Y 333.629,Z 342.549,A -85,B 0,C 180,E1 -14622.501,E2 -14622.501} C_VEL
LIN {X 0,Y 333.594,Z 342.559,A -85,B 0,C 180,E1 -14625.956,E2 -14625.956} C_VEL
LIN {X 0,Y 333.646,Z 342.551,A -85,B 0,C 180,E1 -14629.317,E2 -14629.317} C_VEL
LIN {X 0,Y 333.657,Z 342.665,A -85,B 0,C 180,E1 -14631.12,E2 -14631.12} C_VEL
LIN {X 0,Y 335.51,Z 349.495,A -85,B 0,C 180,E1 -14633.332,E2 -14633.332} C_VEL
LIN {X 0,Y 345.166,Z 369.047,A -85,B 0,C 180,E1 -14634.849,E2 -14634.849} C_VEL
LIN {X 0,Y 352.187,Z 384.935,A -85,B 0,C 180,E1 -14635.924,E2 -14635.924} C_VEL
LIN {X 0,Y 349.355,Z 485.656,A -85,B 0,C 180,E1 -14638.02,E2 -14638.02} C_VEL
LIN {X 0,Y 348.531,Z 500.085,A -85,B 0,C 180,E1 -14638.551,E2 -14638.551} C_VEL
LIN {X 0,Y 347.34,Z 513.697,A -85,B 0,C 180,E1 -14639.277,E2 -14639.277} C_VEL
LIN {X 0,Y 345.697,Z 527.842,A -85,B 0,C 180,E1 -14640.295,E2 -14640.295} C_VEL
LIN {X 0,Y 344.065,Z 540.118,A -85,B 0,C 180,E1 -14641.443,E2 -14641.443} C_VEL
LIN {X 0,Y 342.052,Z 551.895,A -85,B 0,C 180,E1 -14642.797,E2 -14642.797} C_VEL
LIN {X 0,Y 340.263,Z 562.402,A -85,B 0,C 180,E1 -14644.295,E2 -14644.295} C_VEL
LIN {X 0,Y 338.629,Z 571.937,A -85,B 0,C 180,E1 -14645.951,E2 -14645.951} C_VEL
LIN {X 0,Y 337.113,Z 580.021,A -85,B 0,C 180,E1 -14647.638,E2 -14647.638} C_VEL
LIN {X 0,Y 335.699,Z 587.337,A -85,B 0,C 180,E1 -14649.472,E2 -14649.472} C_VEL
LIN {X 0,Y 334.411,Z 594.307,A -85,B 0,C 180,E1 -14651.625,E2 -14651.625} C_VEL
LIN {X 0,Y 333.524,Z 599.106,A -85,B 0,C 180,E1 -14653.473,E2 -14653.473} C_VEL
LIN {X 0,Y 332.929,Z 602.98,A -85,B 0,C 180,E1 -14655.327,E2 -14655.327} C_VEL
LIN {X 0,Y 332.604,Z 605.045,A -85,B 0,C 180,E1 -14656.56,E2 -14656.56} C_VEL
LIN {X 0,Y 332.088,Z 608.081,A -85,B 0,C 180,E1 -14659.02,E2 -14659.02} C_VEL
LIN {X 0,Y 331.938,Z 609.732,A -85,B 0,C 180,E1 -14661.477,E2 -14661.477} C_VEL
LIN {X 0,Y 331.994,Z 610.047,A -85,B 0,C 180,E1 -14663.924,E2 -14663.924} C_VEL
LIN {X 0,Y 332.005,Z 609.048,A -85,B 0,C 180,E1 -14666.359,E2 -14666.359} C_VEL
LIN {X 0,Y 332.065,Z 606.722,A -85,B 0,C 180,E1 -14668.787,E2 -14668.787} C_VEL
LIN {X 0,Y 332.399,Z 603.011,A -85,B 0,C 180,E1 -14671.211,E2 -14671.211} C_VEL
LIN {X 0,Y 332.909,Z 597.803,A -85,B 0,C 180,E1 -14673.631,E2 -14673.631} C_VEL
LIN {X 0,Y 333.548,Z 592.761,A -85,B 0,C 180,E1 -14675.441,E2 -14675.441} C_VEL
LIN {X 0,Y 334.659,Z 585.566,A -85,B 0,C 180,E1 -14677.542,E2 -14677.542} C_VEL
LIN {X 0,Y 335.634,Z 578.05,A -85,B 0,C 180,E1 -14679.339,E2 -14679.339} C_VEL
LIN {X 0,Y 336.847,Z 569.605,A -85,B 0,C 180,E1 -14681.018,E2 -14681.018} C_VEL
LIN {X 0,Y 338.175,Z 560.051,A -85,B 0,C 180,E1 -14682.604,E2 -14682.604} C_VEL
LIN {X 0,Y 339.657,Z 549.34,A -85,B 0,C 180,E1 -14684.071,E2 -14684.071} C_VEL
LIN {X 0,Y 341.08,Z 537.638,A -85,B 0,C 180,E1 -14685.384,E2 -14685.384} C_VEL
LIN {X 0,Y 342.516,Z 524.73,A -85,B 0,C 180,E1 -14686.54,E2 -14686.54} C_VEL
LIN {X 0,Y 343.783,Z 511.216,A -85,B 0,C 180,E1 -14687.473,E2 -14687.473} C_VEL
LIN {X 0,Y 344.737,Z 497.861,A -85,B 0,C 180,E1 -14688.151,E2 -14688.151} C_VEL
LIN {X 0,Y 345.391,Z 483.062,A -85,B 0,C 180,E1 -14688.653,E2 -14688.653} C_VEL
LIN {X 0,Y 347.479,Z 390.681,A -85,B 0,C 180,E1 -14690.57,E2 -14690.57} C_VEL
LIN {X 0,Y 347.066,Z 386.869,A -85,B 0,C 180,E1 -14690.685,E2 -14690.685} C_VEL
LIN {X 0,Y 345.902,Z 383.269,A -85,B 0,C 180,E1 -14690.854,E2 -14690.854} C_VEL
LIN {X 0,Y 343.244,Z 378.268,A -85,B 0,C 180,E1 -14691.171,E2 -14691.171} C_VEL
LIN {X 0,Y 335.742,Z 367.063,A -85,B 0,C 180,E1 -14692.03,E2 -14692.03} C_VEL
LIN {X 0,Y 334.062,Z 363.534,A -85,B 0,C 180,E1 -14692.252,E2 -14692.252} C_VEL
LIN {X 0,Y 327.965,Z 349.045,A -85,B 0,C 180,E1 -14693.159,E2 -14693.159} C_VEL
LIN {X 0,Y 326.697,Z 343.416,A -85,B 0,C 180,E1 -14694.873,E2 -14694.873} C_VEL
LIN {X 0,Y 326.652,Z 343.417,A -85,B 0,C 180,E1 -14698.25,E2 -14698.25} C_VEL
LIN {X 0,Y 326.591,Z 343.428,A -85,B 0,C 180,E1 -14701.094,E2 -14701.094} C_VEL
LIN {X 0,Y 326.608,Z 343.425,A -85,B 0,C 180,E1 -14704.018,E2 -14704.018} C_VEL
LIN {X 0,Y 326.629,Z 343.422,A -85,B 0,C 180,E1 -14707.238,E2 -14707.238} C_VEL
LIN {X 0,Y 326.576,Z 343.414,A -85,B 0,C 180,E1 -14711.13,E2 -14711.13} C_VEL
LIN {X 0,Y 326.525,Z 343.432,A -85,B 0,C 180,E1 -14714.741,E2 -14714.741} C_VEL
LIN {X 0,Y 326.573,Z 343.423,A -85,B 0,C 180,E1 -14718.153,E2 -14718.153} C_VEL
LIN {X 0,Y 326.593,Z 343.424,A -85,B 0,C 180,E1 -14721.386,E2 -14721.386} C_VEL
LIN {X 0,Y 326.615,Z 343.426,A -85,B 0,C 180,E1 -14724.85,E2 -14724.85} C_VEL
LIN {X 0,Y 326.602,Z 343.423,A -85,B 0,C 180,E1 -14727.454,E2 -14727.454} C_VEL
LIN {X 0,Y 326.641,Z 343.419,A -85,B 0,C 180,E1 -14730.338,E2 -14730.338} C_VEL
LIN {X 0,Y 326.662,Z 343.405,A -85,B 0,C 180,E1 -14733.14,E2 -14733.14} C_VEL
LIN {X 0,Y 326.636,Z 343.421,A -85,B 0,C 180,E1 -14735.869,E2 -14735.869} C_VEL
LIN {X 0,Y 326.606,Z 343.407,A -85,B 0,C 180,E1 -14739.861,E2 -14739.861} C_VEL
LIN {X 0,Y 326.7,Z 343.412,A -85,B 0,C 180,E1 -14743.76,E2 -14743.76} C_VEL
LIN {X 0,Y 326.748,Z 343.395,A -85,B 0,C 180,E1 -14746.314,E2 -14746.314} C_VEL
LIN {X 0,Y 326.773,Z 343.4,A -85,B 0,C 180,E1 -14750.092,E2 -14750.092} C_VEL
LIN {X 0,Y 326.947,Z 343.375,A -85,B 0,C 180,E1 -14753.83,E2 -14753.83} C_VEL
LIN {X 0,Y 327.003,Z 343.369,A -85,B 0,C 180,E1 -14757.536,E2 -14757.536} C_VEL
LIN {X 0,Y 327.031,Z 343.368,A -85,B 0,C 180,E1 -14761.231,E2 -14761.231} C_VEL
LIN {X 0,Y 326.928,Z 343.387,A -85,B 0,C 180,E1 -14766.17,E2 -14766.17} C_VEL
LIN {X 0,Y 326.772,Z 343.392,A -85,B 0,C 180,E1 -14769.907,E2 -14769.907} C_VEL
LIN {X 0,Y 326.747,Z 343.408,A -85,B 0,C 180,E1 -14773.686,E2 -14773.686} C_VEL
LIN {X 0,Y 326.654,Z 343.416,A -85,B 0,C 180,E1 -14777.53,E2 -14777.53} C_VEL
LIN {X 0,Y 326.618,Z 343.417,A -85,B 0,C 180,E1 -14780.138,E2 -14780.138} C_VEL
LIN {X 0,Y 326.624,Z 343.423,A -85,B 0,C 180,E1 -14784.131,E2 -14784.131} C_VEL
LIN {X 0,Y 326.595,Z 343.428,A -85,B 0,C 180,E1 -14788.084,E2 -14788.084} C_VEL
LIN {X 0,Y 326.564,Z 343.426,A -85,B 0,C 180,E1 -14791.098,E2 -14791.098} C_VEL
LIN {X 0,Y 326.599,Z 343.424,A -85,B 0,C 180,E1 -14794.02,E2 -14794.02} C_VEL
LIN {X 0,Y 326.62,Z 343.422,A -85,B 0,C 180,E1 -14797.239,E2 -14797.239} C_VEL
LIN {X 0,Y 326.571,Z 343.418,A -85,B 0,C 180,E1 -14801.132,E2 -14801.132} C_VEL
LIN {X 0,Y 326.521,Z 343.435,A -85,B 0,C 180,E1 -14804.743,E2 -14804.743} C_VEL
LIN {X 0,Y 326.571,Z 343.431,A -85,B 0,C 180,E1 -14808.155,E2 -14808.155} C_VEL
LIN {X 0,Y 326.619,Z 343.43,A -85,B 0,C 180,E1 -14811.392,E2 -14811.392} C_VEL
LIN {X 0,Y 326.645,Z 343.485,A -85,B 0,C 180,E1 -14815.333,E2 -14815.333} C_VEL
LIN {X 0,Y 329.642,Z 356.117,A -85,B 0,C 180,E1 -14818.826,E2 -14818.826} C_VEL
LIN {X 0,Y 331.689,Z 365.444,A -85,B 0,C 180,E1 -14821.23,E2 -14821.23} C_VEL
LIN {X 0,Y 335.114,Z 375.016,A -85,B 0,C 180,E1 -14821.741,E2 -14821.741} C_VEL
LIN {X 0,Y 338.962,Z 397.714,A -85,B 0,C 180,E1 -14822.575,E2 -14822.575} C_VEL
LIN {X 0,Y 340.672,Z 408.981,A -85,B 0,C 180,E1 -14822.964,E2 -14822.964} C_VEL
LIN {X 0,Y 338.368,Z 503.393,A -85,B 0,C 180,E1 -14824.964,E2 -14824.964} C_VEL
LIN {X 0,Y 337.454,Z 518.071,A -85,B 0,C 180,E1 -14825.508,E2 -14825.508} C_VEL
LIN {X 0,Y 336.281,Z 532.094,A -85,B 0,C 180,E1 -14826.278,E2 -14826.278} C_VEL
LIN {X 0,Y 334.842,Z 546.027,A -85,B 0,C 180,E1 -14827.316,E2 -14827.316} C_VEL
LIN {X 0,Y 333.301,Z 558.489,A -85,B 0,C 180,E1 -14828.509,E2 -14828.509} C_VEL
LIN {X 0,Y 331.737,Z 569.89,A -85,B 0,C 180,E1 -14829.864,E2 -14829.864} C_VEL
LIN {X 0,Y 330.197,Z 580.368,A -85,B 0,C 180,E1 -14831.382,E2 -14831.382} C_VEL
LIN {X 0,Y 328.653,Z 590.788,A -85,B 0,C 180,E1 -14833.221,E2 -14833.221} C_VEL
LIN {X 0,Y 327.489,Z 599.39,A -85,B 0,C 180,E1 -14835.077,E2 -14835.077} C_VEL
LIN {X 0,Y 326.474,Z 607.597,A -85,B 0,C 180,E1 -14837.253,E2 -14837.253} C_VEL
LIN {X 0,Y 325.615,Z 614.198,A -85,B 0,C 180,E1 -14839.429,E2 -14839.429} C_VEL
LIN {X 0,Y 325.149,Z 620.053,A -85,B 0,C 180,E1 -14841.924,E2 -14841.924} C_VEL
LIN {X 0,Y 324.976,Z 623.939,A -85,B 0,C 180,E1 -14844.156,E2 -14844.156} C_VEL
LIN {X 0,Y 324.895,Z 626.549,A -85,B 0,C 180,E1 -14846.279,E2 -14846.279} C_VEL
LIN {X 0,Y 324.835,Z 628.295,A -85,B 0,C 180,E1 -14848.76,E2 -14848.76} C_VEL
LIN {X 0,Y 324.874,Z 628.665,A -85,B 0,C 180,E1 -14850,E2 -14850} C_VEL
LIN {X 0,Y 324.83,Z 628.398,A -85,B 0,C 180,E1 -14852.48,E2 -14852.48} C_VEL
LIN {X 0,Y 324.873,Z 626.798,A -85,B 0,C 180,E1 -14854.964,E2 -14854.964} C_VEL
LIN {X 0,Y 325.111,Z 623.837,A -85,B 0,C 180,E1 -14857.452,E2 -14857.452} C_VEL
LIN {X 0,Y 325.579,Z 619.435,A -85,B 0,C 180,E1 -14859.944,E2 -14859.944} C_VEL
LIN {X 0,Y 326.528,Z 613.472,A -85,B 0,C 180,E1 -14862.429,E2 -14862.429} C_VEL
LIN {X 0,Y 327.677,Z 606.778,A -85,B 0,C 180,E1 -14864.596,E2 -14864.596} C_VEL
LIN {X 0,Y 329.155,Z 598.468,A -85,B 0,C 180,E1 -14866.753,E2 -14866.753} C_VEL
LIN {X 0,Y 330.842,Z 589.83,A -85,B 0,C 180,E1 -14868.58,E2 -14868.58} C_VEL
LIN {X 0,Y 332.902,Z 579.382,A -85,B 0,C 180,E1 -14870.385,E2 -14870.385} C_VEL
LIN {X 0,Y 334.846,Z 568.884,A -85,B 0,C 180,E1 -14871.872,E2 -14871.872} C_VEL
LIN {X 0,Y 336.929,Z 556.056,A -85,B 0,C 180,E1 -14873.348,E2 -14873.348} C_VEL
LIN {X 0,Y 338.774,Z 543.234,A -85,B 0,C 180,E1 -14874.513,E2 -14874.513} C_VEL
LIN {X 0,Y 340.443,Z 529.908,A -85,B 0,C 180,E1 -14875.444,E2 -14875.444} C_VEL
LIN {X 0,Y 341.859,Z 516.143,A -85,B 0,C 180,E1 -14876.149,E2 -14876.149} C_VEL
LIN {X 0,Y 342.846,Z 501.767,A -85,B 0,C 180,E1 -14876.641,E2 -14876.641} C_VEL
LIN {X 0,Y 345.419,Z 409.535,A -85,B 0,C 180,E1 -14878.597,E2 -14878.597} C_VEL
LIN {X 0,Y 340.811,Z 385.195,A -85,B 0,C 180,E1 -14879.649,E2 -14879.649} C_VEL
LIN {X 0,Y 339.587,Z 381.185,A -85,B 0,C 180,E1 -14879.876,E2 -14879.876} C_VEL
LIN {X 0,Y 332.05,Z 364.655,A -85,B 0,C 180,E1 -14881.147,E2 -14881.147} C_VEL
LIN {X 0,Y 329.349,Z 353.429,A -85,B 0,C 180,E1 -14884.434,E2 -14884.434} C_VEL
LIN {X 0,Y 326.617,Z 343.412,A -85,B 0,C 180,E1 -14887.586,E2 -14887.586} C_VEL
LIN {X 0,Y 326.573,Z 343.415,A -85,B 0,C 180,E1 -14891.13,E2 -14891.13} C_VEL
LIN {X 0,Y 326.522,Z 343.429,A -85,B 0,C 180,E1 -14894.742,E2 -14894.742} C_VEL
LIN {X 0,Y 326.57,Z 343.428,A -85,B 0,C 180,E1 -14898.154,E2 -14898.154} C_VEL
LIN {X 0,Y 326.617,Z 343.425,A -85,B 0,C 180,E1 -14901.391,E2 -14901.391} C_VEL
LIN {X 0,Y 326.612,Z 343.421,A -85,B 0,C 180,E1 -14904.851,E2 -14904.851} C_VEL
LIN {X 0,Y 326.6,Z 343.427,A -85,B 0,C 180,E1 -14907.455,E2 -14907.455} C_VEL
LIN {X 0,Y 326.582,Z 343.401,A -85,B 0,C 180,E1 -14910.333,E2 -14910.333} C_VEL
LIN {X 0,Y 326.626,Z 343.419,A -85,B 0,C 180,E1 -14914.511,E2 -14914.511} C_VEL
LIN {X 0,Y 326.605,Z 343.422,A -85,B 0,C 180,E1 -14918.543,E2 -14918.543} C_VEL
LIN {X 0,Y 326.699,Z 343.413,A -85,B 0,C 180,E1 -14921.175,E2 -14921.175} C_VEL
LIN {X 0,Y 326.754,Z 343.406,A -85,B 0,C 180,E1 -14925.434,E2 -14925.434} C_VEL
LIN {X 0,Y 326.743,Z 343.4,A -85,B 0,C 180,E1 -14928.838,E2 -14928.838} C_VEL
LIN {X 0,Y 326.903,Z 343.381,A -85,B 0,C 180,E1 -14932.589,E2 -14932.589} C_VEL
LIN {X 0,Y 326.738,Z 343.409,A -85,B 0,C 180,E1 -14935.065,E2 -14935.065} C_VEL
LIN {X 0,Y 326.999,Z 343.368,A -85,B 0,C 180,E1 -14937.537,E2 -14937.537} C_VEL
LIN {X 0,Y 327.019,Z 343.373,A -85,B 0,C 180,E1 -14941.232,E2 -14941.232} C_VEL
LIN {X 0,Y 326.757,Z 343.403,A -85,B 0,C 180,E1 -14943.7,E2 -14943.7} C_VEL
LIN {X 0,Y 326.918,Z 343.38,A -85,B 0,C 180,E1 -14946.578,E2 -14946.578} C_VEL
LIN {X 0,Y 326.774,Z 343.405,A -85,B 0,C 180,E1 -14949.908,E2 -14949.908} C_VEL
LIN {X 0,Y 326.75,Z 343.408,A -85,B 0,C 180,E1 -14953.686,E2 -14953.686} C_VEL
LIN {X 0,Y 326.656,Z 343.418,A -85,B 0,C 180,E1 -14957.531,E2 -14957.531} C_VEL
LIN {X 0,Y 326.61,Z 343.423,A -85,B 0,C 180,E1 -14961.458,E2 -14961.458} C_VEL
LIN {X 0,Y 326.684,Z 343.416,A -85,B 0,C 180,E1 -14965.485,E2 -14965.485} C_VEL
LIN {X 0,Y 326.642,Z 343.421,A -85,B 0,C 180,E1 -14969.662,E2 -14969.662} C_VEL
LIN {X 0,Y 326.602,Z 343.423,A -85,B 0,C 180,E1 -14974.021,E2 -14974.021} C_VEL
LIN {X 0,Y 326.623,Z 343.418,A -85,B 0,C 180,E1 -14977.24,E2 -14977.24} C_VEL
LIN {X 0,Y 326.575,Z 343.431,A -85,B 0,C 180,E1 -14981.132,E2 -14981.132} C_VEL
LIN {X 0,Y 326.525,Z 343.435,A -85,B 0,C 180,E1 -14984.744,E2 -14984.744} C_VEL
LIN {X 0,Y 326.575,Z 343.432,A -85,B 0,C 180,E1 -14988.155,E2 -14988.155} C_VEL
LIN {X 0,Y 326.58,Z 343.448,A -85,B 0,C 180,E1 -14990.404,E2 -14990.404} C_VEL
LIN {X 0,Y 328.285,Z 349.753,A -85,B 0,C 180,E1 -14992.505,E2 -14992.505} C_VEL
LIN {X 0,Y 336.198,Z 365.143,A -85,B 0,C 180,E1 -14993.8,E2 -14993.8} C_VEL
LIN {X 0,Y 345.21,Z 384.792,A -85,B 0,C 180,E1 -14995.231,E2 -14995.231} C_VEL
LIN {X 0,Y 346.111,Z 387.636,A -85,B 0,C 180,E1 -14995.39,E2 -14995.39} C_VEL
LIN {X 0,Y 343.115,Z 486.32,A -85,B 0,C 180,E1 -14997.473,E2 -14997.473} C_VEL
LIN {X 0,Y 342.204,Z 501.027,A -85,B 0,C 180,E1 -14998.031,E2 -14998.031} C_VEL
LIN {X 0,Y 340.934,Z 515.025,A -85,B 0,C 180,E1 -14998.808,E2 -14998.808} C_VEL
LIN {X 0,Y 339.237,Z 528.923,A -85,B 0,C 180,E1 -14999.843,E2 -14999.843} C_VEL
LIN {X 0,Y 337.316,Z 542.004,A -85,B 0,C 180,E1 -15001.105,E2 -15001.105} C_VEL
LIN {X 0,Y 335.227,Z 553.803,A -85,B 0,C 180,E1 -15002.534,E2 -15002.534} C_VEL
LIN {X 0,Y 333.402,Z 564.018,A -85,B 0,C 180,E1 -15004.063,E2 -15004.063} C_VEL
LIN {X 0,Y 331.7,Z 573.583,A -85,B 0,C 180,E1 -15005.808,E2 -15005.808} C_VEL
LIN {X 0,Y 329.895,Z 582.492,A -85,B 0,C 180,E1 -15007.782,E2 -15007.782} C_VEL
LIN {X 0,Y 328.298,Z 590.452,A -85,B 0,C 180,E1 -15009.97,E2 -15009.97} C_VEL
LIN {X 0,Y 327.213,Z 596.013,A -85,B 0,C 180,E1 -15011.855,E2 -15011.855} C_VEL
LIN {X 0,Y 326.137,Z 601.816,A -85,B 0,C 180,E1 -15014.374,E2 -15014.374} C_VEL
LIN {X 0,Y 325.614,Z 605.132,A -85,B 0,C 180,E1 -15016.266,E2 -15016.266} C_VEL
LIN {X 0,Y 325.053,Z 608.211,A -85,B 0,C 180,E1 -15018.78,E2 -15018.78} C_VEL
LIN {X 0,Y 324.843,Z 609.904,A -85,B 0,C 180,E1 -15021.29,E2 -15021.29} C_VEL
LIN {X 0,Y 324.888,Z 610.26,A -85,B 0,C 180,E1 -15023.791,E2 -15023.791} C_VEL
LIN {X 0,Y 324.93,Z 609.301,A -85,B 0,C 180,E1 -15026.28,E2 -15026.28} C_VEL
LIN {X 0,Y 324.965,Z 607.018,A -85,B 0,C 180,E1 -15028.761,E2 -15028.761} C_VEL
LIN {X 0,Y 325.322,Z 603.349,A -85,B 0,C 180,E1 -15031.238,E2 -15031.238} C_VEL
LIN {X 0,Y 325.848,Z 598.197,A -85,B 0,C 180,E1 -15033.71,E2 -15033.71} C_VEL
LIN {X 0,Y 326.521,Z 593.194,A -85,B 0,C 180,E1 -15035.558,E2 -15035.558} C_VEL
LIN {X 0,Y 327.652,Z 586.053,A -85,B 0,C 180,E1 -15037.704,E2 -15037.704} C_VEL
LIN {X 0,Y 328.666,Z 578.597,A -85,B 0,C 180,E1 -15039.539,E2 -15039.539} C_VEL
LIN {X 0,Y 329.763,Z 571.257,A -85,B 0,C 180,E1 -15041.058,E2 -15041.058} C_VEL
LIN {X 0,Y 331.308,Z 560.747,A -85,B 0,C 180,E1 -15042.869,E2 -15042.869} C_VEL
LIN {X 0,Y 332.829,Z 550.138,A -85,B 0,C 180,E1 -15044.365,E2 -15044.365} C_VEL
LIN {X 0,Y 334.297,Z 538.564,A -85,B 0,C 180,E1 -15045.704,E2 -15045.704} C_VEL
LIN {X 0,Y 335.777,Z 525.827,A -85,B 0,C 180,E1 -15046.882,E2 -15046.882} C_VEL
LIN {X 0,Y 337.09,Z 512.591,A -85,B 0,C 180,E1 -15047.831,E2 -15047.831} C_VEL
LIN {X 0,Y 338.082,Z 498.949,A -85,B 0,C 180,E1 -15048.56,E2 -15048.56} C_VEL
LIN {X 0,Y 338.762,Z 484.836,A -85,B 0,C 180,E1 -15049.071,E2 -15049.071} C_VEL
LIN {X 0,Y 341.055,Z 382.735,A -85,B 0,C 180,E1 -15051.241,E2 -15051.241} C_VEL
LIN {X 0,Y 339.458,Z 377.36,A -85,B 0,C 180,E1 -15051.49,E2 -15051.49} C_VEL
LIN {X 0,Y 334.062,Z 363.534,A -85,B 0,C 180,E1 -15052.252,E2 -15052.252} C_VEL
LIN {X 0,Y 332.745,Z 362.052,A -85,B 0,C 180,E1 -15052.398,E2 -15052.398} C_VEL
LIN {X 0,Y 325.905,Z 359.815,A -85,B 0,C 180,E1 -15053.045,E2 -15053.045} C_VEL
LIN {X 0,Y 324.781,Z 358.56,A -85,B 0,C 180,E1 -15053.175,E2 -15053.175} C_VEL
LIN {X 0,Y 320.79,Z 349.296,A -85,B 0,C 180,E1 -15053.798,E2 -15053.798} C_VEL
LIN {X 0,Y 319.668,Z 344.293,A -85,B 0,C 180,E1 -15055.387,E2 -15055.387} C_VEL
LIN {X 0,Y 319.581,Z 344.295,A -85,B 0,C 180,E1 -15058.933,E2 -15058.933} C_VEL
LIN {X 0,Y 319.532,Z 344.31,A -85,B 0,C 180,E1 -15061.861,E2 -15061.861} C_VEL
LIN {X 0,Y 319.58,Z 344.292,A -85,B 0,C 180,E1 -15065.542,E2 -15065.542} C_VEL
LIN {X 0,Y 319.573,Z 344.302,A -85,B 0,C 180,E1 -15068.007,E2 -15068.007} C_VEL
LIN {X 0,Y 319.524,Z 344.297,A -85,B 0,C 180,E1 -15071.596,E2 -15071.596} C_VEL
LIN {X 0,Y 319.486,Z 344.31,A -85,B 0,C 180,E1 -15075.256,E2 -15075.256} C_VEL
LIN {X 0,Y 319.525,Z 344.301,A -85,B 0,C 180,E1 -15078.71,E2 -15078.71} C_VEL
LIN {X 0,Y 319.549,Z 344.297,A -85,B 0,C 180,E1 -15082.349,E2 -15082.349} C_VEL
LIN {X 0,Y 319.556,Z 344.305,A -85,B 0,C 180,E1 -15085.122,E2 -15085.122} C_VEL
LIN {X 0,Y 319.561,Z 344.306,A -85,B 0,C 180,E1 -15089.058,E2 -15089.058} C_VEL
LIN {X 0,Y 319.589,Z 344.284,A -85,B 0,C 180,E1 -15092.496,E2 -15092.496} C_VEL
LIN {X 0,Y 319.58,Z 344.303,A -85,B 0,C 180,E1 -15095.301,E2 -15095.301} C_VEL
LIN {X 0,Y 319.557,Z 344.297,A -85,B 0,C 180,E1 -15098.044,E2 -15098.044} C_VEL
LIN {X 0,Y 319.606,Z 344.293,A -85,B 0,C 180,E1 -15102.069,E2 -15102.069} C_VEL
LIN {X 0,Y 319.722,Z 344.273,A -85,B 0,C 180,E1 -15106.007,E2 -15106.007} C_VEL
LIN {X 0,Y 319.726,Z 344.278,A -85,B 0,C 180,E1 -15109.871,E2 -15109.871} C_VEL
LIN {X 0,Y 319.905,Z 344.252,A -85,B 0,C 180,E1 -15113.693,E2 -15113.693} C_VEL
LIN {X 0,Y 319.949,Z 344.248,A -85,B 0,C 180,E1 -15117.482,E2 -15117.482} C_VEL
LIN {X 0,Y 319.998,Z 344.243,A -85,B 0,C 180,E1 -15121.258,E2 -15121.258} C_VEL
LIN {X 0,Y 319.886,Z 344.265,A -85,B 0,C 180,E1 -15126.306,E2 -15126.306} C_VEL
LIN {X 0,Y 319.724,Z 344.271,A -85,B 0,C 180,E1 -15130.128,E2 -15130.128} C_VEL
LIN {X 0,Y 319.721,Z 344.282,A -85,B 0,C 180,E1 -15133.992,E2 -15133.992} C_VEL
LIN {X 0,Y 319.615,Z 344.295,A -85,B 0,C 180,E1 -15137.929,E2 -15137.929} C_VEL
LIN {X 0,Y 319.557,Z 344.293,A -85,B 0,C 180,E1 -15141.955,E2 -15141.955} C_VEL
LIN {X 0,Y 319.563,Z 344.295,A -85,B 0,C 180,E1 -15146.094,E2 -15146.094} C_VEL
LIN {X 0,Y 319.535,Z 344.304,A -85,B 0,C 180,E1 -15148.939,E2 -15148.939} C_VEL
LIN {X 0,Y 319.516,Z 344.309,A -85,B 0,C 180,E1 -15151.863,E2 -15151.863} C_VEL
LIN {X 0,Y 319.572,Z 344.302,A -85,B 0,C 180,E1 -15155.543,E2 -15155.543} C_VEL
LIN {X 0,Y 319.55,Z 344.304,A -85,B 0,C 180,E1 -15158.011,E2 -15158.011} C_VEL
LIN {X 0,Y 319.519,Z 344.295,A -85,B 0,C 180,E1 -15161.598,E2 -15161.598} C_VEL
LIN {X 0,Y 319.482,Z 344.312,A -85,B 0,C 180,E1 -15165.258,E2 -15165.258} C_VEL
LIN {X 0,Y 319.523,Z 344.309,A -85,B 0,C 180,E1 -15168.712,E2 -15168.712} C_VEL
LIN {X 0,Y 319.557,Z 344.31,A -85,B 0,C 180,E1 -15172.349,E2 -15172.349} C_VEL
LIN {X 0,Y 319.584,Z 344.416,A -85,B 0,C 180,E1 -15174.836,E2 -15174.836} C_VEL
LIN {X 0,Y 322.434,Z 356.287,A -85,B 0,C 180,E1 -15178.219,E2 -15178.219} C_VEL
LIN {X 0,Y 324.362,Z 365.068,A -85,B 0,C 180,E1 -15180.583,E2 -15180.583} C_VEL
LIN {X 0,Y 328.89,Z 377.032,A -85,B 0,C 180,E1 -15181.267,E2 -15181.267} C_VEL
LIN {X 0,Y 332.585,Z 399.125,A -85,B 0,C 180,E1 -15182.098,E2 -15182.098} C_VEL
LIN {X 0,Y 334.227,Z 409.387,A -85,B 0,C 180,E1 -15182.47,E2 -15182.47} C_VEL
LIN {X 0,Y 331.868,Z 502.8,A -85,B 0,C 180,E1 -15184.481,E2 -15184.481} C_VEL
LIN {X 0,Y 331.007,Z 516.861,A -85,B 0,C 180,E1 -15184.999,E2 -15184.999} C_VEL
LIN {X 0,Y 329.751,Z 531.14,A -85,B 0,C 180,E1 -15185.779,E2 -15185.779} C_VEL
LIN {X 0,Y 328.44,Z 543.455,A -85,B 0,C 180,E1 -15186.681,E2 -15186.681} C_VEL
LIN {X 0,Y 326.775,Z 556.884,A -85,B 0,C 180,E1 -15187.95,E2 -15187.95} C_VEL
LIN {X 0,Y 325.183,Z 568.113,A -85,B 0,C 180,E1 -15189.274,E2 -15189.274} C_VEL
LIN {X 0,Y 323.673,Z 577.87,A -85,B 0,C 180,E1 -15190.663,E2 -15190.663} C_VEL
LIN {X 0,Y 322.032,Z 588.682,A -85,B 0,C 180,E1 -15192.538,E2 -15192.538} C_VEL
LIN {X 0,Y 320.75,Z 597.744,A -85,B 0,C 180,E1 -15194.464,E2 -15194.464} C_VEL
LIN {X 0,Y 319.731,Z 605.018,A -85,B 0,C 180,E1 -15196.332,E2 -15196.332} C_VEL
LIN {X 0,Y 318.778,Z 612.101,A -85,B 0,C 180,E1 -15198.556,E2 -15198.556} C_VEL
LIN {X 0,Y 318.173,Z 618.457,A -85,B 0,C 180,E1 -15201.105,E2 -15201.105} C_VEL
LIN {X 0,Y 317.903,Z 623.137,A -85,B 0,C 180,E1 -15203.654,E2 -15203.654} C_VEL
LIN {X 0,Y 317.803,Z 626.302,A -85,B 0,C 180,E1 -15206.196,E2 -15206.196} C_VEL
LIN {X 0,Y 317.746,Z 628.075,A -85,B 0,C 180,E1 -15208.733,E2 -15208.733} C_VEL
LIN {X 0,Y 317.781,Z 628.457,A -85,B 0,C 180,E1 -15210,E2 -15210} C_VEL
LIN {X 0,Y 317.751,Z 628.216,A -85,B 0,C 180,E1 -15212.535,E2 -15212.535} C_VEL
LIN {X 0,Y 317.789,Z 626.641,A -85,B 0,C 180,E1 -15215.075,E2 -15215.075} C_VEL
LIN {X 0,Y 318.03,Z 623.706,A -85,B 0,C 180,E1 -15217.619,E2 -15217.619} C_VEL
LIN {X 0,Y 318.543,Z 619.332,A -85,B 0,C 180,E1 -15220.166,E2 -15220.166} C_VEL
LIN {X 0,Y 319.549,Z 613.403,A -85,B 0,C 180,E1 -15222.705,E2 -15222.705} C_VEL
LIN {X 0,Y 320.781,Z 606.747,A -85,B 0,C 180,E1 -15224.917,E2 -15224.917} C_VEL
LIN {X 0,Y 322.333,Z 598.488,A -85,B 0,C 180,E1 -15227.118,E2 -15227.118} C_VEL
LIN {X 0,Y 324.104,Z 589.896,A -85,B 0,C 180,E1 -15228.981,E2 -15228.981} C_VEL
LIN {X 0,Y 326.246,Z 579.501,A -85,B 0,C 180,E1 -15230.82,E2 -15230.82} C_VEL
LIN {X 0,Y 328.264,Z 569.069,A -85,B 0,C 180,E1 -15232.334,E2 -15232.334} C_VEL
LIN {X 0,Y 330.233,Z 557.67,A -85,B 0,C 180,E1 -15233.692,E2 -15233.692} C_VEL
LIN {X 0,Y 332.112,Z 545.378,A -85,B 0,C 180,E1 -15234.871,E2 -15234.871} C_VEL
LIN {X 0,Y 333.932,Z 531.581,A -85,B 0,C 180,E1 -15235.893,E2 -15235.893} C_VEL
LIN {X 0,Y 335.466,Z 517.724,A -85,B 0,C 180,E1 -15236.644,E2 -15236.644} C_VEL
LIN {X 0,Y 336.563,Z 503.305,A -85,B 0,C 180,E1 -15237.179,E2 -15237.179} C_VEL
LIN {X 0,Y 339.418,Z 411.622,A -85,B 0,C 180,E1 -15239.151,E2 -15239.151} C_VEL
LIN {X 0,Y 336.092,Z 392.873,A -85,B 0,C 180,E1 -15239.96,E2 -15239.96} C_VEL
LIN {X 0,Y 334.251,Z 384.936,A -85,B 0,C 180,E1 -15240.357,E2 -15240.357} C_VEL
LIN {X 0,Y 326.735,Z 368.563,A -85,B 0,C 180,E1 -15241.628,E2 -15241.628} C_VEL
LIN {X 0,Y 324.773,Z 364.418,A -85,B 0,C 180,E1 -15242.004,E2 -15242.004} C_VEL
LIN {X 0,Y 322.131,Z 353.518,A -85,B 0,C 180,E1 -15245.312,E2 -15245.312} C_VEL
LIN {X 0,Y 319.591,Z 344.292,A -85,B 0,C 180,E1 -15248.355,E2 -15248.355} C_VEL
LIN {X 0,Y 319.521,Z 344.298,A -85,B 0,C 180,E1 -15251.596,E2 -15251.596} C_VEL
LIN {X 0,Y 319.482,Z 344.305,A -85,B 0,C 180,E1 -15255.256,E2 -15255.256} C_VEL
LIN {X 0,Y 319.522,Z 344.308,A -85,B 0,C 180,E1 -15258.711,E2 -15258.711} C_VEL
LIN {X 0,Y 319.555,Z 344.302,A -85,B 0,C 180,E1 -15262.347,E2 -15262.347} C_VEL
LIN {X 0,Y 319.552,Z 344.299,A -85,B 0,C 180,E1 -15265.123,E2 -15265.123} C_VEL
LIN {X 0,Y 319.516,Z 344.299,A -85,B 0,C 180,E1 -15268.137,E2 -15268.137} C_VEL
LIN {X 0,Y 319.562,Z 344.287,A -85,B 0,C 180,E1 -15271.604,E2 -15271.604} C_VEL
LIN {X 0,Y 319.565,Z 344.296,A -85,B 0,C 180,E1 -15275.301,E2 -15275.301} C_VEL
LIN {X 0,Y 319.557,Z 344.303,A -85,B 0,C 180,E1 -15278.045,E2 -15278.045} C_VEL
LIN {X 0,Y 319.615,Z 344.296,A -85,B 0,C 180,E1 -15282.071,E2 -15282.071} C_VEL
LIN {X 0,Y 319.72,Z 344.285,A -85,B 0,C 180,E1 -15286.008,E2 -15286.008} C_VEL
LIN {X 0,Y 319.723,Z 344.283,A -85,B 0,C 180,E1 -15289.872,E2 -15289.872} C_VEL
LIN {X 0,Y 319.889,Z 344.255,A -85,B 0,C 180,E1 -15293.694,E2 -15293.694} C_VEL
LIN {X 0,Y 319.945,Z 344.247,A -85,B 0,C 180,E1 -15297.482,E2 -15297.482} C_VEL
LIN {X 0,Y 319.988,Z 344.248,A -85,B 0,C 180,E1 -15301.259,E2 -15301.259} C_VEL
LIN {X 0,Y 319.707,Z 344.282,A -85,B 0,C 180,E1 -15303.782,E2 -15303.782} C_VEL
LIN {X 0,Y 319.882,Z 344.258,A -85,B 0,C 180,E1 -15306.565,E2 -15306.565} C_VEL
LIN {X 0,Y 319.726,Z 344.282,A -85,B 0,C 180,E1 -15310.129,E2 -15310.129} C_VEL
LIN {X 0,Y 319.724,Z 344.283,A -85,B 0,C 180,E1 -15313.993,E2 -15313.993} C_VEL
LIN {X 0,Y 319.606,Z 344.297,A -85,B 0,C 180,E1 -15317.93,E2 -15317.93} C_VEL
LIN {X 0,Y 319.561,Z 344.302,A -85,B 0,C 180,E1 -15321.955,E2 -15321.955} C_VEL
LIN {X 0,Y 319.628,Z 344.295,A -85,B 0,C 180,E1 -15326.089,E2 -15326.089} C_VEL
LIN {X 0,Y 319.574,Z 344.3,A -85,B 0,C 180,E1 -15328.936,E2 -15328.936} C_VEL
LIN {X 0,Y 319.525,Z 344.302,A -85,B 0,C 180,E1 -15331.863,E2 -15331.863} C_VEL
LIN {X 0,Y 319.575,Z 344.3,A -85,B 0,C 180,E1 -15335.544,E2 -15335.544} C_VEL
LIN {X 0,Y 319.553,Z 344.3,A -85,B 0,C 180,E1 -15338.012,E2 -15338.012} C_VEL
LIN {X 0,Y 319.523,Z 344.309,A -85,B 0,C 180,E1 -15341.598,E2 -15341.598} C_VEL
LIN {X 0,Y 319.486,Z 344.313,A -85,B 0,C 180,E1 -15345.258,E2 -15345.258} C_VEL
LIN {X 0,Y 319.527,Z 344.307,A -85,B 0,C 180,E1 -15348.713,E2 -15348.713} C_VEL
LIN {X 0,Y 319.562,Z 344.43,A -85,B 0,C 180,E1 -15349.718,E2 -15349.718} C_VEL
LIN {X 0,Y 321.048,Z 349.874,A -85,B 0,C 180,E1 -15351.626,E2 -15351.626} C_VEL
LIN {X 0,Y 330.556,Z 368.114,A -85,B 0,C 180,E1 -15353.242,E2 -15353.242} C_VEL
LIN {X 0,Y 339.758,Z 388.33,A -85,B 0,C 180,E1 -15354.755,E2 -15354.755} C_VEL
LIN {X 0,Y 339.986,Z 390.79,A -85,B 0,C 180,E1 -15354.839,E2 -15354.839} C_VEL
LIN {X 0,Y 336.925,Z 486.62,A -85,B 0,C 180,E1 -15356.893,E2 -15356.893} C_VEL
LIN {X 0,Y 335.986,Z 501.216,A -85,B 0,C 180,E1 -15357.455,E2 -15357.455} C_VEL
LIN {X 0,Y 334.66,Z 515.214,A -85,B 0,C 180,E1 -15358.244,E2 -15358.244} C_VEL
LIN {X 0,Y 333.013,Z 528.218,A -85,B 0,C 180,E1 -15359.219,E2 -15359.219} C_VEL
LIN {X 0,Y 331.308,Z 539.972,A -85,B 0,C 180,E1 -15360.347,E2 -15360.347} C_VEL
LIN {X 0,Y 329.022,Z 552.273,A -85,B 0,C 180,E1 -15361.798,E2 -15361.798} C_VEL
LIN {X 0,Y 326.923,Z 563.756,A -85,B 0,C 180,E1 -15363.509,E2 -15363.509} C_VEL
LIN {X 0,Y 324.952,Z 574.076,A -85,B 0,C 180,E1 -15365.426,E2 -15365.426} C_VEL
LIN {X 0,Y 323.18,Z 582.377,A -85,B 0,C 180,E1 -15367.295,E2 -15367.295} C_VEL
LIN {X 0,Y 321.481,Z 590.395,A -85,B 0,C 180,E1 -15369.527,E2 -15369.527} C_VEL
LIN {X 0,Y 320.331,Z 596.008,A -85,B 0,C 180,E1 -15371.451,E2 -15371.451} C_VEL
LIN {X 0,Y 319.159,Z 601.859,A -85,B 0,C 180,E1 -15374.023,E2 -15374.023} C_VEL
LIN {X 0,Y 318.559,Z 605.423,A -85,B 0,C 180,E1 -15376.104,E2 -15376.104} C_VEL
LIN {X 0,Y 317.995,Z 608.342,A -85,B 0,C 180,E1 -15378.527,E2 -15378.527} C_VEL
LIN {X 0,Y 317.763,Z 610.076,A -85,B 0,C 180,E1 -15381.094,E2 -15381.094} C_VEL
LIN {X 0,Y 317.798,Z 610.473,A -85,B 0,C 180,E1 -15383.652,E2 -15383.652} C_VEL
LIN {X 0,Y 317.834,Z 609.554,A -85,B 0,C 180,E1 -15386.196,E2 -15386.196} C_VEL
LIN {X 0,Y 317.868,Z 607.312,A -85,B 0,C 180,E1 -15388.733,E2 -15388.733} C_VEL
LIN {X 0,Y 318.231,Z 603.686,A -85,B 0,C 180,E1 -15391.265,E2 -15391.265} C_VEL
LIN {X 0,Y 318.774,Z 598.581,A -85,B 0,C 180,E1 -15393.792,E2 -15393.792} C_VEL
LIN {X 0,Y 319.495,Z 593.624,A -85,B 0,C 180,E1 -15395.681,E2 -15395.681} C_VEL
LIN {X 0,Y 320.646,Z 586.538,A -85,B 0,C 180,E1 -15397.873,E2 -15397.873} C_VEL
LIN {X 0,Y 321.704,Z 579.142,A -85,B 0,C 180,E1 -15399.747,E2 -15399.747} C_VEL
LIN {X 0,Y 322.978,Z 570.799,A -85,B 0,C 180,E1 -15401.505,E2 -15401.505} C_VEL
LIN {X 0,Y 324.43,Z 561.442,A -85,B 0,C 180,E1 -15403.147,E2 -15403.147} C_VEL
LIN {X 0,Y 326.189,Z 549.766,A -85,B 0,C 180,E1 -15404.824,E2 -15404.824} C_VEL
LIN {X 0,Y 327.698,Z 538.072,A -85,B 0,C 180,E1 -15406.188,E2 -15406.188} C_VEL
LIN {X 0,Y 329.232,Z 525.17,A -85,B 0,C 180,E1 -15407.388,E2 -15407.388} C_VEL
LIN {X 0,Y 330.589,Z 511.669,A -85,B 0,C 180,E1 -15408.354,E2 -15408.354} C_VEL
LIN {X 0,Y 331.625,Z 498.334,A -85,B 0,C 180,E1 -15409.056,E2 -15409.056} C_VEL
LIN {X 0,Y 332.321,Z 483.583,A -85,B 0,C 180,E1 -15409.576,E2 -15409.576} C_VEL
LIN {X 0,Y 334.699,Z 384.211,A -85,B 0,C 180,E1 -15411.716,E2 -15411.716} C_VEL
LIN {X 0,Y 330.515,Z 372.304,A -85,B 0,C 180,E1 -15412.345,E2 -15412.345} C_VEL
LIN {X 0,Y 324.781,Z 358.56,A -85,B 0,C 180,E1 -15413.175,E2 -15413.175} C_VEL
LIN {X 0,Y 322.637,Z 355.425,A -85,B 0,C 180,E1 -15413.447,E2 -15413.447} C_VEL
LIN {X 0,Y 319.928,Z 352.931,A -85,B 0,C 180,E1 -15413.784,E2 -15413.784} C_VEL
LIN {X 0,Y 315.469,Z 349.586,A -85,B 0,C 180,E1 -15414.509,E2 -15414.509} C_VEL
LIN {X 0,Y 313.519,Z 347.702,A -85,B 0,C 180,E1 -15415.06,E2 -15415.06} C_VEL
LIN {X 0,Y 312.859,Z 346.402,A -85,B 0,C 180,E1 -15415.472,E2 -15415.472} C_VEL
LIN {X 0,Y 312.605,Z 345.172,A -85,B 0,C 180,E1 -15415.934,E2 -15415.934} C_VEL
LIN {X 0,Y 312.539,Z 345.176,A -85,B 0,C 180,E1 -15419.65,E2 -15419.65} C_VEL
LIN {X 0,Y 312.52,Z 345.183,A -85,B 0,C 180,E1 -15423.688,E2 -15423.688} C_VEL
LIN {X 0,Y 312.538,Z 345.178,A -85,B 0,C 180,E1 -15427.382,E2 -15427.382} C_VEL
LIN {X 0,Y 312.489,Z 345.166,A -85,B 0,C 180,E1 -15430.708,E2 -15430.708} C_VEL
LIN {X 0,Y 312.449,Z 345.186,A -85,B 0,C 180,E1 -15434.208,E2 -15434.208} C_VEL
LIN {X 0,Y 312.481,Z 345.179,A -85,B 0,C 180,E1 -15437.917,E2 -15437.917} C_VEL
LIN {X 0,Y 312.494,Z 345.186,A -85,B 0,C 180,E1 -15440.97,E2 -15440.97} C_VEL
LIN {X 0,Y 312.527,Z 345.179,A -85,B 0,C 180,E1 -15444.219,E2 -15444.219} C_VEL
LIN {X 0,Y 312.499,Z 345.178,A -85,B 0,C 180,E1 -15447.333,E2 -15447.333} C_VEL
LIN {X 0,Y 312.535,Z 345.168,A -85,B 0,C 180,E1 -15451.279,E2 -15451.279} C_VEL
LIN {X 0,Y 312.554,Z 345.172,A -85,B 0,C 180,E1 -15454.708,E2 -15454.708} C_VEL
LIN {X 0,Y 312.513,Z 345.165,A -85,B 0,C 180,E1 -15458.91,E2 -15458.91} C_VEL
LIN {X 0,Y 312.57,Z 345.176,A -85,B 0,C 180,E1 -15463.004,E2 -15463.004} C_VEL
LIN {X 0,Y 312.676,Z 345.151,A -85,B 0,C 180,E1 -15465.685,E2 -15465.685} C_VEL
LIN {X 0,Y 312.676,Z 345.156,A -85,B 0,C 180,E1 -15469.64,E2 -15469.64} C_VEL
LIN {X 0,Y 312.819,Z 345.143,A -85,B 0,C 180,E1 -15472.252,E2 -15472.252} C_VEL
LIN {X 0,Y 312.688,Z 345.138,A -85,B 0,C 180,E1 -15474.841,E2 -15474.841} C_VEL
LIN {X 0,Y 312.957,Z 345.126,A -85,B 0,C 180,E1 -15478.713,E2 -15478.713} C_VEL
LIN {X 0,Y 312.965,Z 345.119,A -85,B 0,C 180,E1 -15481.286,E2 -15481.286} C_VEL
LIN {X 0,Y 312.828,Z 345.145,A -85,B 0,C 180,E1 -15486.449,E2 -15486.449} C_VEL
LIN {X 0,Y 312.741,Z 345.139,A -85,B 0,C 180,E1 -15489.05,E2 -15489.05} C_VEL
LIN {X 0,Y 312.622,Z 345.167,A -85,B 0,C 180,E1 -15492.991,E2 -15492.991} C_VEL
LIN {X 0,Y 312.612,Z 345.157,A -85,B 0,C 180,E1 -15495.651,E2 -15495.651} C_VEL
LIN {X 0,Y 312.549,Z 345.175,A -85,B 0,C 180,E1 -15499.712,E2 -15499.712} C_VEL
LIN {X 0,Y 312.514,Z 345.181,A -85,B 0,C 180,E1 -15503.878,E2 -15503.878} C_VEL
LIN {X 0,Y 312.489,Z 345.178,A -85,B 0,C 180,E1 -15506.731,E2 -15506.731} C_VEL
LIN {X 0,Y 312.487,Z 345.181,A -85,B 0,C 180,E1 -15509.656,E2 -15509.656} C_VEL
LIN {X 0,Y 312.512,Z 345.179,A -85,B 0,C 180,E1 -15513.689,E2 -15513.689} C_VEL
LIN {X 0,Y 312.519,Z 345.178,A -85,B 0,C 180,E1 -15517.386,E2 -15517.386} C_VEL
LIN {X 0,Y 312.483,Z 345.175,A -85,B 0,C 180,E1 -15520.71,E2 -15520.71} C_VEL
LIN {X 0,Y 312.446,Z 345.189,A -85,B 0,C 180,E1 -15524.21,E2 -15524.21} C_VEL
LIN {X 0,Y 312.479,Z 345.188,A -85,B 0,C 180,E1 -15527.919,E2 -15527.919} C_VEL
LIN {X 0,Y 312.501,Z 345.189,A -85,B 0,C 180,E1 -15531.918,E2 -15531.918} C_VEL
LIN {X 0,Y 312.57,Z 345.367,A -85,B 0,C 180,E1 -15534.326,E2 -15534.326} C_VEL
LIN {X 0,Y 315.654,Z 358.283,A -85,B 0,C 180,E1 -15538.101,E2 -15538.101} C_VEL
LIN {X 0,Y 317.155,Z 364.969,A -85,B 0,C 180,E1 -15539.921,E2 -15539.921} C_VEL
LIN {X 0,Y 322.801,Z 379.648,A -85,B 0,C 180,E1 -15540.799,E2 -15540.799} C_VEL
LIN {X 0,Y 326.356,Z 401.255,A -85,B 0,C 180,E1 -15541.63,E2 -15541.63} C_VEL
LIN {X 0,Y 327.766,Z 411.173,A -85,B 0,C 180,E1 -15541.985,E2 -15541.985} C_VEL
LIN {X 0,Y 325.327,Z 503.39,A -85,B 0,C 180,E1 -15544.016,E2 -15544.016} C_VEL
LIN {X 0,Y 324.407,Z 517.167,A -85,B 0,C 180,E1 -15544.54,E2 -15544.54} C_VEL
LIN {X 0,Y 323.113,Z 531.315,A -85,B 0,C 180,E1 -15545.334,E2 -15545.334} C_VEL
LIN {X 0,Y 321.681,Z 544.435,A -85,B 0,C 180,E1 -15546.332,E2 -15546.332} C_VEL
LIN {X 0,Y 320.091,Z 556.79,A -85,B 0,C 180,E1 -15547.534,E2 -15547.534} C_VEL
LIN {X 0,Y 318.314,Z 568.703,A -85,B 0,C 180,E1 -15548.975,E2 -15548.975} C_VEL
LIN {X 0,Y 316.61,Z 579.312,A -85,B 0,C 180,E1 -15550.552,E2 -15550.552} C_VEL
LIN {X 0,Y 314.956,Z 589.853,A -85,B 0,C 180,E1 -15552.468,E2 -15552.468} C_VEL
LIN {X 0,Y 313.595,Z 598.987,A -85,B 0,C 180,E1 -15554.509,E2 -15554.509} C_VEL
LIN {X 0,Y 312.526,Z 606.859,A -85,B 0,C 180,E1 -15556.674,E2 -15556.674} C_VEL
LIN {X 0,Y 311.549,Z 613.527,A -85,B 0,C 180,E1 -15558.946,E2 -15558.946} C_VEL
LIN {X 0,Y 311.004,Z 619.445,A -85,B 0,C 180,E1 -15561.554,E2 -15561.554} C_VEL
LIN {X 0,Y 310.826,Z 622.859,A -85,B 0,C 180,E1 -15563.509,E2 -15563.509} C_VEL
LIN {X 0,Y 310.715,Z 626.054,A -85,B 0,C 180,E1 -15566.109,E2 -15566.109} C_VEL
LIN {X 0,Y 310.66,Z 627.854,A -85,B 0,C 180,E1 -15568.704,E2 -15568.704} C_VEL
LIN {X 0,Y 310.691,Z 628.249,A -85,B 0,C 180,E1 -15570,E2 -15570} C_VEL
LIN {X 0,Y 310.673,Z 628.034,A -85,B 0,C 180,E1 -15572.593,E2 -15572.593} C_VEL
LIN {X 0,Y 310.695,Z 626.485,A -85,B 0,C 180,E1 -15575.191,E2 -15575.191} C_VEL
LIN {X 0,Y 310.977,Z 623.577,A -85,B 0,C 180,E1 -15577.793,E2 -15577.793} C_VEL
LIN {X 0,Y 311.524,Z 619.232,A -85,B 0,C 180,E1 -15580.397,E2 -15580.397} C_VEL
LIN {X 0,Y 312.588,Z 613.333,A -85,B 0,C 180,E1 -15582.993,E2 -15582.993} C_VEL
LIN {X 0,Y 313.897,Z 606.713,A -85,B 0,C 180,E1 -15585.252,E2 -15585.252} C_VEL
LIN {X 0,Y 315.518,Z 598.51,A -85,B 0,C 180,E1 -15587.499,E2 -15587.499} C_VEL
LIN {X 0,Y 317.376,Z 589.962,A -85,B 0,C 180,E1 -15589.399,E2 -15589.399} C_VEL
LIN {X 0,Y 319.591,Z 579.625,A -85,B 0,C 180,E1 -15591.274,E2 -15591.274} C_VEL
LIN {X 0,Y 321.926,Z 568.089,A -85,B 0,C 180,E1 -15592.968,E2 -15592.968} C_VEL
LIN {X 0,Y 323.957,Z 556.6,A -85,B 0,C 180,E1 -15594.342,E2 -15594.342} C_VEL
LIN {X 0,Y 325.942,Z 544.006,A -85,B 0,C 180,E1 -15595.546,E2 -15595.546} C_VEL
LIN {X 0,Y 327.731,Z 531.011,A -85,B 0,C 180,E1 -15596.507,E2 -15596.507} C_VEL
LIN {X 0,Y 329.329,Z 517.027,A -85,B 0,C 180,E1 -15597.267,E2 -15597.267} C_VEL
LIN {X 0,Y 330.465,Z 502.337,A -85,B 0,C 180,E1 -15597.809,E2 -15597.809} C_VEL
LIN {X 0,Y 333.282,Z 411.812,A -85,B 0,C 180,E1 -15599.791,E2 -15599.791} C_VEL
LIN {X 0,Y 328.91,Z 388.606,A -85,B 0,C 180,E1 -15600.86,E2 -15600.86} C_VEL
LIN {X 0,Y 321.807,Z 372.885,A -85,B 0,C 180,E1 -15602.105,E2 -15602.105} C_VEL
LIN {X 0,Y 317.59,Z 364.404,A -85,B 0,C 180,E1 -15602.856,E2 -15602.856} C_VEL
LIN {X 0,Y 315.273,Z 355.105,A -85,B 0,C 180,E1 -15605.757,E2 -15605.757} C_VEL
LIN {X 0,Y 312.519,Z 345.172,A -85,B 0,C 180,E1 -15609.124,E2 -15609.124} C_VEL
LIN {X 0,Y 312.485,Z 345.179,A -85,B 0,C 180,E1 -15612.431,E2 -15612.431} C_VEL
LIN {X 0,Y 312.452,Z 345.185,A -85,B 0,C 180,E1 -15616.034,E2 -15616.034} C_VEL
LIN {X 0,Y 312.498,Z 345.18,A -85,B 0,C 180,E1 -15619.874,E2 -15619.874} C_VEL
LIN {X 0,Y 312.528,Z 345.181,A -85,B 0,C 180,E1 -15624.05,E2 -15624.05} C_VEL
LIN {X 0,Y 312.494,Z 345.184,A -85,B 0,C 180,E1 -15627.333,E2 -15627.333} C_VEL
LIN {X 0,Y 312.492,Z 345.162,A -85,B 0,C 180,E1 -15631.294,E2 -15631.294} C_VEL
LIN {X 0,Y 312.539,Z 345.173,A -85,B 0,C 180,E1 -15634.707,E2 -15634.707} C_VEL
LIN {X 0,Y 312.554,Z 345.178,A -85,B 0,C 180,E1 -15637.527,E2 -15637.527} C_VEL
LIN {X 0,Y 312.573,Z 345.177,A -85,B 0,C 180,E1 -15641.653,E2 -15641.653} C_VEL
LIN {X 0,Y 312.675,Z 345.163,A -85,B 0,C 180,E1 -15645.686,E2 -15645.686} C_VEL
LIN {X 0,Y 312.673,Z 345.158,A -85,B 0,C 180,E1 -15649.641,E2 -15649.641} C_VEL
LIN {X 0,Y 312.786,Z 345.14,A -85,B 0,C 180,E1 -15652.253,E2 -15652.253} C_VEL
LIN {X 0,Y 312.678,Z 345.159,A -85,B 0,C 180,E1 -15654.842,E2 -15654.842} C_VEL
LIN {X 0,Y 312.971,Z 345.117,A -85,B 0,C 180,E1 -15658.714,E2 -15658.714} C_VEL
LIN {X 0,Y 312.901,Z 345.122,A -85,B 0,C 180,E1 -15662.575,E2 -15662.575} C_VEL
LIN {X 0,Y 312.836,Z 345.137,A -85,B 0,C 180,E1 -15666.547,E2 -15666.547} C_VEL
LIN {X 0,Y 312.742,Z 345.151,A -85,B 0,C 180,E1 -15669.051,E2 -15669.051} C_VEL
LIN {X 0,Y 312.625,Z 345.16,A -85,B 0,C 180,E1 -15672.992,E2 -15672.992} C_VEL
LIN {X 0,Y 312.614,Z 345.163,A -85,B 0,C 180,E1 -15675.652,E2 -15675.652} C_VEL
LIN {X 0,Y 312.532,Z 345.175,A -85,B 0,C 180,E1 -15679.714,E2 -15679.714} C_VEL
LIN {X 0,Y 312.52,Z 345.184,A -85,B 0,C 180,E1 -15682.781,E2 -15682.781} C_VEL
LIN {X 0,Y 312.596,Z 345.171,A -85,B 0,C 180,E1 -15685.936,E2 -15685.936} C_VEL
LIN {X 0,Y 312.533,Z 345.179,A -85,B 0,C 180,E1 -15689.652,E2 -15689.652} C_VEL
LIN {X 0,Y 312.515,Z 345.179,A -85,B 0,C 180,E1 -15693.69,E2 -15693.69} C_VEL
LIN {X 0,Y 312.521,Z 345.174,A -85,B 0,C 180,E1 -15697.386,E2 -15697.386} C_VEL
LIN {X 0,Y 312.487,Z 345.183,A -85,B 0,C 180,E1 -15700.71,E2 -15700.71} C_VEL
LIN {X 0,Y 312.449,Z 345.19,A -85,B 0,C 180,E1 -15704.211,E2 -15704.211} C_VEL
LIN {X 0,Y 312.483,Z 345.189,A -85,B 0,C 180,E1 -15707.92,E2 -15707.92} C_VEL
LIN {X 0,Y 312.509,Z 345.282,A -85,B 0,C 180,E1 -15708.947,E2 -15708.947} C_VEL
LIN {X 0,Y 313.883,Z 350.276,A -85,B 0,C 180,E1 -15710.712,E2 -15710.712} C_VEL
LIN {X 0,Y 323.984,Z 369.131,A -85,B 0,C 180,E1 -15712.497,E2 -15712.497} C_VEL
LIN {X 0,Y 332.396,Z 387.343,A -85,B 0,C 180,E1 -15713.936,E2 -15713.936} C_VEL
LIN {X 0,Y 333.916,Z 390.913,A -85,B 0,C 180,E1 -15714.193,E2 -15714.193} C_VEL
LIN {X 0,Y 330.795,Z 486.561,A -85,B 0,C 180,E1 -15716.279,E2 -15716.279} C_VEL
LIN {X 0,Y 329.896,Z 500.649,A -85,B 0,C 180,E1 -15716.823,E2 -15716.823} C_VEL
LIN {X 0,Y 328.578,Z 514.27,A -85,B 0,C 180,E1 -15717.585,E2 -15717.585} C_VEL
LIN {X 0,Y 326.869,Z 527.523,A -85,B 0,C 180,E1 -15718.575,E2 -15718.575} C_VEL
LIN {X 0,Y 325.06,Z 539.284,A -85,B 0,C 180,E1 -15719.698,E2 -15719.698} C_VEL
LIN {X 0,Y 322.703,Z 551.902,A -85,B 0,C 180,E1 -15721.198,E2 -15721.198} C_VEL
LIN {X 0,Y 320.864,Z 561.503,A -85,B 0,C 180,E1 -15722.616,E2 -15722.616} C_VEL
LIN {X 0,Y 319.024,Z 570.501,A -85,B 0,C 180,E1 -15724.203,E2 -15724.203} C_VEL
LIN {X 0,Y 317.173,Z 579.582,A -85,B 0,C 180,E1 -15726.148,E2 -15726.148} C_VEL
LIN {X 0,Y 315.175,Z 588.204,A -85,B 0,C 180,E1 -15728.413,E2 -15728.413} C_VEL
LIN {X 0,Y 313.852,Z 594.215,A -85,B 0,C 180,E1 -15730.374,E2 -15730.374} C_VEL
LIN {X 0,Y 312.789,Z 599.164,A -85,B 0,C 180,E1 -15732.343,E2 -15732.343} C_VEL
LIN {X 0,Y 311.766,Z 604.243,A -85,B 0,C 180,E1 -15734.976,E2 -15734.976} C_VEL
LIN {X 0,Y 311.234,Z 607.069,A -85,B 0,C 180,E1 -15736.95,E2 -15736.95} C_VEL
LIN {X 0,Y 310.751,Z 609.53,A -85,B 0,C 180,E1 -15739.576,E2 -15739.576} C_VEL
LIN {X 0,Y 310.68,Z 610.632,A -85,B 0,C 180,E1 -15742.199,E2 -15742.199} C_VEL
LIN {X 0,Y 310.715,Z 610.41,A -85,B 0,C 180,E1 -15744.809,E2 -15744.809} C_VEL
LIN {X 0,Y 310.735,Z 608.874,A -85,B 0,C 180,E1 -15747.407,E2 -15747.407} C_VEL
LIN {X 0,Y 310.92,Z 605.992,A -85,B 0,C 180,E1 -15750,E2 -15750} C_VEL
LIN {X 0,Y 311.354,Z 601.688,A -85,B 0,C 180,E1 -15752.587,E2 -15752.587} C_VEL
LIN {X 0,Y 312.122,Z 595.83,A -85,B 0,C 180,E1 -15755.167,E2 -15755.167} C_VEL
LIN {X 0,Y 313.228,Z 589.227,A -85,B 0,C 180,E1 -15757.412,E2 -15757.412} C_VEL
LIN {X 0,Y 314.606,Z 581.019,A -85,B 0,C 180,E1 -15759.645,E2 -15759.645} C_VEL
LIN {X 0,Y 316.067,Z 571.41,A -85,B 0,C 180,E1 -15761.76,E2 -15761.76} C_VEL
LIN {X 0,Y 317.558,Z 562.134,A -85,B 0,C 180,E1 -15763.437,E2 -15763.437} C_VEL
LIN {X 0,Y 319.364,Z 550.558,A -85,B 0,C 180,E1 -15765.148,E2 -15765.148} C_VEL
LIN {X 0,Y 320.946,Z 538.986,A -85,B 0,C 180,E1 -15766.539,E2 -15766.539} C_VEL
LIN {X 0,Y 322.523,Z 526.254,A -85,B 0,C 180,E1 -15767.762,E2 -15767.762} C_VEL
LIN {X 0,Y 323.945,Z 513.019,A -85,B 0,C 180,E1 -15768.744,E2 -15768.744} C_VEL
LIN {X 0,Y 325.006,Z 499.388,A -85,B 0,C 180,E1 -15769.5,E2 -15769.5} C_VEL
LIN {X 0,Y 325.738,Z 485.307,A -85,B 0,C 180,E1 -15770.029,E2 -15770.029} C_VEL
LIN {X 0,Y 328.274,Z 385.267,A -85,B 0,C 180,E1 -15772.227,E2 -15772.227} C_VEL
LIN {X 0,Y 321.483,Z 367.693,A -85,B 0,C 180,E1 -15773.249,E2 -15773.249} C_VEL
LIN {X 0,Y 314.398,Z 351.641,A -85,B 0,C 180,E1 -15774.315,E2 -15774.315} C_VEL
LIN {X 0,Y 313.609,Z 349.516,A -85,B 0,C 180,E1 -15774.475,E2 -15774.475} C_VEL
LIN {X 0,Y 312.859,Z 346.402,A -85,B 0,C 180,E1 -15775.472,E2 -15775.472} C_VEL
LIN {X 0,Y 312.373,Z 345.516,A -85,B 0,C 180,E1 -15775.951,E2 -15775.951} C_VEL
LIN {X 0,Y 311.129,Z 345.355,A -85,B 0,C 180,E1 -15776.797,E2 -15776.797} C_VEL
LIN {X 0,Y 306.422,Z 346.066,A -85,B 0,C 180,E1 -15779.656,E2 -15779.656} C_VEL
LIN {X 0,Y 305.438,Z 346.062,A -85,B 0,C 180,E1 -15781.171,E2 -15781.171} C_VEL
LIN {X 0,Y 305.463,Z 346.051,A -85,B 0,C 180,E1 -15785.112,E2 -15785.112} C_VEL
LIN {X 0,Y 305.467,Z 346.058,A -85,B 0,C 180,E1 -15788.532,E2 -15788.532} C_VEL
LIN {X 0,Y 305.453,Z 346.059,A -85,B 0,C 180,E1 -15792.584,E2 -15792.584} C_VEL
LIN {X 0,Y 305.423,Z 346.064,A -85,B 0,C 180,E1 -15796.344,E2 -15796.344} C_VEL
LIN {X 0,Y 305.455,Z 346.061,A -85,B 0,C 180,E1 -15799.891,E2 -15799.891} C_VEL
LIN {X 0,Y 305.476,Z 346.059,A -85,B 0,C 180,E1 -15803.631,E2 -15803.631} C_VEL
LIN {X 0,Y 305.46,Z 346.053,A -85,B 0,C 180,E1 -15806.482,E2 -15806.482} C_VEL
LIN {X 0,Y 305.452,Z 346.06,A -85,B 0,C 180,E1 -15809.589,E2 -15809.589} C_VEL
LIN {X 0,Y 305.482,Z 346.04,A -85,B 0,C 180,E1 -15812.604,E2 -15812.604} C_VEL
LIN {X 0,Y 305.485,Z 346.057,A -85,B 0,C 180,E1 -15815.536,E2 -15815.536} C_VEL
LIN {X 0,Y 305.474,Z 346.037,A -85,B 0,C 180,E1 -15819.811,E2 -15819.811} C_VEL
LIN {X 0,Y 305.543,Z 346.048,A -85,B 0,C 180,E1 -15823.977,E2 -15823.977} C_VEL
LIN {X 0,Y 305.575,Z 346.026,A -85,B 0,C 180,E1 -15826.703,E2 -15826.703} C_VEL
LIN {X 0,Y 305.747,Z 346.024,A -85,B 0,C 180,E1 -15831.258,E2 -15831.258} C_VEL
LIN {X 0,Y 305.795,Z 346.009,A -85,B 0,C 180,E1 -15833.401,E2 -15833.401} C_VEL
LIN {X 0,Y 305.925,Z 346.002,A -85,B 0,C 180,E1 -15838.683,E2 -15838.683} C_VEL
LIN {X 0,Y 305.932,Z 345.995,A -85,B 0,C 180,E1 -15841.316,E2 -15841.316} C_VEL
LIN {X 0,Y 305.773,Z 346.022,A -85,B 0,C 180,E1 -15846.599,E2 -15846.599} C_VEL
LIN {X 0,Y 305.685,Z 346.017,A -85,B 0,C 180,E1 -15849.261,E2 -15849.261} C_VEL
LIN {X 0,Y 305.575,Z 346.044,A -85,B 0,C 180,E1 -15853.296,E2 -15853.296} C_VEL
LIN {X 0,Y 305.542,Z 346.038,A -85,B 0,C 180,E1 -15856.022,E2 -15856.022} C_VEL
LIN {X 0,Y 305.533,Z 346.048,A -85,B 0,C 180,E1 -15859.426,E2 -15859.426} C_VEL
LIN {X 0,Y 305.478,Z 346.054,A -85,B 0,C 180,E1 -15863.04,E2 -15863.04} C_VEL
LIN {X 0,Y 305.462,Z 346.051,A -85,B 0,C 180,E1 -15866.198,E2 -15866.198} C_VEL
LIN {X 0,Y 305.44,Z 346.06,A -85,B 0,C 180,E1 -15869.034,E2 -15869.034} C_VEL
LIN {X 0,Y 305.429,Z 346.064,A -85,B 0,C 180,E1 -15871.954,E2 -15871.954} C_VEL
LIN {X 0,Y 305.455,Z 346.058,A -85,B 0,C 180,E1 -15875.114,E2 -15875.114} C_VEL
LIN {X 0,Y 305.443,Z 346.062,A -85,B 0,C 180,E1 -15878.529,E2 -15878.529} C_VEL
LIN {X 0,Y 305.449,Z 346.054,A -85,B 0,C 180,E1 -15882.586,E2 -15882.586} C_VEL
LIN {X 0,Y 305.42,Z 346.065,A -85,B 0,C 180,E1 -15886.346,E2 -15886.346} C_VEL
LIN {X 0,Y 305.453,Z 346.064,A -85,B 0,C 180,E1 -15889.893,E2 -15889.893} C_VEL
LIN {X 0,Y 305.495,Z 346.194,A -85,B 0,C 180,E1 -15893.749,E2 -15893.749} C_VEL
LIN {X 0,Y 308.483,Z 358.449,A -85,B 0,C 180,E1 -15897.453,E2 -15897.453} C_VEL
LIN {X 0,Y 309.808,Z 364.544,A -85,B 0,C 180,E1 -15899.203,E2 -15899.203} C_VEL
LIN {X 0,Y 316.606,Z 381.54,A -85,B 0,C 180,E1 -15900.284,E2 -15900.284} C_VEL
LIN {X 0,Y 320.101,Z 403.084,A -85,B 0,C 180,E1 -15901.134,E2 -15901.134} C_VEL
LIN {X 0,Y 321.37,Z 411.51,A -85,B 0,C 180,E1 -15901.451,E2 -15901.451} C_VEL
LIN {X 0,Y 318.85,Z 502.786,A -85,B 0,C 180,E1 -15903.491,E2 -15903.491} C_VEL
LIN {X 0,Y 317.949,Z 516.708,A -85,B 0,C 180,E1 -15904.028,E2 -15904.028} C_VEL
LIN {X 0,Y 316.62,Z 530.347,A -85,B 0,C 180,E1 -15904.793,E2 -15904.793} C_VEL
LIN {X 0,Y 315.139,Z 543.635,A -85,B 0,C 180,E1 -15905.809,E2 -15905.809} C_VEL
LIN {X 0,Y 313.413,Z 556.742,A -85,B 0,C 180,E1 -15907.105,E2 -15907.105} C_VEL
LIN {X 0,Y 311.668,Z 568.105,A -85,B 0,C 180,E1 -15908.505,E2 -15908.505} C_VEL
LIN {X 0,Y 309.857,Z 578.779,A -85,B 0,C 180,E1 -15910.11,E2 -15910.11} C_VEL
LIN {X 0,Y 308.116,Z 589.375,A -85,B 0,C 180,E1 -15912.066,E2 -15912.066} C_VEL
LIN {X 0,Y 306.611,Z 599.148,A -85,B 0,C 180,E1 -15914.302,E2 -15914.302} C_VEL
LIN {X 0,Y 305.542,Z 606.485,A -85,B 0,C 180,E1 -15916.364,E2 -15916.364} C_VEL
LIN {X 0,Y 304.532,Z 613.19,A -85,B 0,C 180,E1 -15918.688,E2 -15918.688} C_VEL
LIN {X 0,Y 303.948,Z 619.139,A -85,B 0,C 180,E1 -15921.356,E2 -15921.356} C_VEL
LIN {X 0,Y 303.738,Z 622.576,A -85,B 0,C 180,E1 -15923.357,E2 -15923.357} C_VEL
LIN {X 0,Y 303.629,Z 625.806,A -85,B 0,C 180,E1 -15926.018,E2 -15926.018} C_VEL
LIN {X 0,Y 303.576,Z 627.633,A -85,B 0,C 180,E1 -15928.674,E2 -15928.674} C_VEL
LIN {X 0,Y 303.603,Z 628.041,A -85,B 0,C 180,E1 -15930,E2 -15930} C_VEL
LIN {X 0,Y 303.598,Z 627.852,A -85,B 0,C 180,E1 -15932.654,E2 -15932.654} C_VEL
LIN {X 0,Y 303.616,Z 626.329,A -85,B 0,C 180,E1 -15935.313,E2 -15935.313} C_VEL
LIN {X 0,Y 303.913,Z 623.448,A -85,B 0,C 180,E1 -15937.975,E2 -15937.975} C_VEL
LIN {X 0,Y 304.512,Z 619.133,A -85,B 0,C 180,E1 -15940.64,E2 -15940.64} C_VEL
LIN {X 0,Y 305.276,Z 614.884,A -85,B 0,C 180,E1 -15942.633,E2 -15942.633} C_VEL
LIN {X 0,Y 306.554,Z 608.697,A -85,B 0,C 180,E1 -15944.946,E2 -15944.946} C_VEL
LIN {X 0,Y 308.136,Z 601.002,A -85,B 0,C 180,E1 -15947.247,E2 -15947.247} C_VEL
LIN {X 0,Y 310.308,Z 591.513,A -85,B 0,C 180,E1 -15949.515,E2 -15949.515} C_VEL
LIN {X 0,Y 312.594,Z 581.589,A -85,B 0,C 180,E1 -15951.428,E2 -15951.428} C_VEL
LIN {X 0,Y 314.964,Z 570.575,A -85,B 0,C 180,E1 -15953.158,E2 -15953.158} C_VEL
LIN {X 0,Y 317.339,Z 557.819,A -85,B 0,C 180,E1 -15954.768,E2 -15954.768} C_VEL
LIN {X 0,Y 319.345,Z 546.164,A -85,B 0,C 180,E1 -15955.937,E2 -15955.937} C_VEL
LIN {X 0,Y 321.132,Z 533.828,A -85,B 0,C 180,E1 -15956.919,E2 -15956.919} C_VEL
LIN {X 0,Y 322.852,Z 520.134,A -85,B 0,C 180,E1 -15957.729,E2 -15957.729} C_VEL
LIN {X 0,Y 324.11,Z 505.974,A -85,B 0,C 180,E1 -15958.315,E2 -15958.315} C_VEL
LIN {X 0,Y 324.939,Z 487.455,A -85,B 0,C 180,E1 -15958.783,E2 -15958.783} C_VEL
LIN {X 0,Y 327.273,Z 412.885,A -85,B 0,C 180,E1 -15960.424,E2 -15960.424} C_VEL
LIN {X 0,Y 323.232,Z 391.31,A -85,B 0,C 180,E1 -15961.448,E2 -15961.448} C_VEL
LIN {X 0,Y 316.009,Z 375.692,A -85,B 0,C 180,E1 -15962.75,E2 -15962.75} C_VEL
LIN {X 0,Y 310.28,Z 364.007,A -85,B 0,C 180,E1 -15963.839,E2 -15963.839} C_VEL
LIN {X 0,Y 307.857,Z 354.481,A -85,B 0,C 180,E1 -15966.965,E2 -15966.965} C_VEL
LIN {X 0,Y 305.47,Z 346.041,A -85,B 0,C 180,E1 -15969.949,E2 -15969.949} C_VEL
LIN {X 0,Y 305.42,Z 346.057,A -85,B 0,C 180,E1 -15973.654,E2 -15973.654} C_VEL
LIN {X 0,Y 305.449,Z 346.055,A -85,B 0,C 180,E1 -15977.414,E2 -15977.414} C_VEL
LIN {X 0,Y 305.469,Z 346.06,A -85,B 0,C 180,E1 -15981.597,E2 -15981.597} C_VEL
LIN {X 0,Y 305.455,Z 346.056,A -85,B 0,C 180,E1 -15984.886,E2 -15984.886} C_VEL
LIN {X 0,Y 305.434,Z 346.049,A -85,B 0,C 180,E1 -15988.358,E2 -15988.358} C_VEL
LIN {X 0,Y 305.457,Z 346.035,A -85,B 0,C 180,E1 -15991.108,E2 -15991.108} C_VEL
LIN {X 0,Y 305.492,Z 346.054,A -85,B 0,C 180,E1 -15994.081,E2 -15994.081} C_VEL
LIN {X 0,Y 305.465,Z 346.056,A -85,B 0,C 180,E1 -15998.401,E2 -15998.401} C_VEL
LIN {X 0,Y 305.534,Z 346.05,A -85,B 0,C 180,E1 -16001.214,E2 -16001.214} C_VEL
LIN {X 0,Y 305.617,Z 346.039,A -85,B 0,C 180,E1 -16005.348,E2 -16005.348} C_VEL
LIN {X 0,Y 305.612,Z 346.035,A -85,B 0,C 180,E1 -16009.399,E2 -16009.399} C_VEL
LIN {X 0,Y 305.736,Z 346.019,A -85,B 0,C 180,E1 -16012.073,E2 -16012.073} C_VEL
LIN {X 0,Y 305.648,Z 346.034,A -85,B 0,C 180,E1 -16014.723,E2 -16014.723} C_VEL
LIN {X 0,Y 305.938,Z 345.993,A -85,B 0,C 180,E1 -16018.684,E2 -16018.684} C_VEL
LIN {X 0,Y 305.926,Z 345.998,A -85,B 0,C 180,E1 -16021.317,E2 -16021.317} C_VEL
LIN {X 0,Y 305.659,Z 346.038,A -85,B 0,C 180,E1 -16025.278,E2 -16025.278} C_VEL
LIN {X 0,Y 305.753,Z 346.015,A -85,B 0,C 180,E1 -16027.928,E2 -16027.928} C_VEL
LIN {X 0,Y 305.589,Z 346.032,A -85,B 0,C 180,E1 -16031.946,E2 -16031.946} C_VEL
LIN {X 0,Y 305.601,Z 346.042,A -85,B 0,C 180,E1 -16035.015,E2 -16035.015} C_VEL
LIN {X 0,Y 305.51,Z 346.056,A -85,B 0,C 180,E1 -16038.788,E2 -16038.788} C_VEL
LIN {X 0,Y 305.48,Z 346.058,A -85,B 0,C 180,E1 -16043.04,E2 -16043.04} C_VEL
LIN {X 0,Y 305.526,Z 346.052,A -85,B 0,C 180,E1 -16046.222,E2 -16046.222} C_VEL
LIN {X 0,Y 305.483,Z 346.056,A -85,B 0,C 180,E1 -16049.048,E2 -16049.048} C_VEL
LIN {X 0,Y 305.437,Z 346.057,A -85,B 0,C 180,E1 -16051.954,E2 -16051.954} C_VEL
LIN {X 0,Y 305.458,Z 346.056,A -85,B 0,C 180,E1 -16055.115,E2 -16055.115} C_VEL
LIN {X 0,Y 305.446,Z 346.061,A -85,B 0,C 180,E1 -16058.53,E2 -16058.53} C_VEL
LIN {X 0,Y 305.452,Z 346.058,A -85,B 0,C 180,E1 -16062.587,E2 -16062.587} C_VEL
LIN {X 0,Y 305.424,Z 346.065,A -85,B 0,C 180,E1 -16066.346,E2 -16066.346} C_VEL
LIN {X 0,Y 305.452,Z 346.193,A -85,B 0,C 180,E1 -16068.146,E2 -16068.146} C_VEL
LIN {X 0,Y 306.666,Z 350.528,A -85,B 0,C 180,E1 -16069.732,E2 -16069.732} C_VEL
LIN {X 0,Y 308.942,Z 354.536,A -85,B 0,C 180,E1 -16070.164,E2 -16070.164} C_VEL
LIN {X 0,Y 318.279,Z 371.977,A -85,B 0,C 180,E1 -16071.873,E2 -16071.873} C_VEL
LIN {X 0,Y 326.026,Z 388.687,A -85,B 0,C 180,E1 -16073.249,E2 -16073.249} C_VEL
LIN {X 0,Y 327.852,Z 392.915,A -85,B 0,C 180,E1 -16073.568,E2 -16073.568} C_VEL
LIN {X 0,Y 324.682,Z 486.966,A -85,B 0,C 180,E1 -16075.657,E2 -16075.657} C_VEL
LIN {X 0,Y 323.682,Z 501.631,A -85,B 0,C 180,E1 -16076.242,E2 -16076.242} C_VEL
LIN {X 0,Y 322.242,Z 515.622,A -85,B 0,C 180,E1 -16077.053,E2 -16077.053} C_VEL
LIN {X 0,Y 320.477,Z 528.624,A -85,B 0,C 180,E1 -16078.059,E2 -16078.059} C_VEL
LIN {X 0,Y 318.453,Z 541.22,A -85,B 0,C 180,E1 -16079.314,E2 -16079.314} C_VEL
LIN {X 0,Y 316.169,Z 552.674,A -85,B 0,C 180,E1 -16080.724,E2 -16080.724} C_VEL
